REGION Network 2: WatchDog WinCC- PLC
   RUNG wire#powerrail
      Contact( "AlwaysTRUE" )
      Contact( "IEC_Timer_WatchDogWicc-PLC_DB".Q )
      wire#w1
      { S7_Templates := "DestType := Int" } Inc( "Dane_ComunicationControlHMI".tempWatchDog_WinCC )
   END_RUNG
   RUNG wire#powerrail
      Contact( "IEC_Timer_WatchDogWinCC_cd_DB".Q )
   END_RUNG wire#w1
   RUNG wire#powerrail
      { S7_Templates := "SrcType := Int" } GE_Contact(in1 := "Dane_ComunicationControlHMI".tempWatchDog_WinCC, in2 := 70)
      P_Trig( "memRis_Foult_WiCC_PLC" )
      S_Coil( "dbmanagement".sterowanie_1.alarm_comunication_WinCC )
   END_RUNG
   // the same network as SCL:
   IF ("AlwaysTRUE" AND "IEC_Timer_WatchDogWicc-PLC_DB".Q) OR "IEC_Timer_WatchDogWinCC_cd_DB".Q THEN
       "Dane_ComunicationControlHMI".tempWatchDog_WinCC := "Dane_ComunicationControlHMI".tempWatchDog_WinCC + 1;
   END_IF;
   #_w1 := "Dane_ComunicationControlHMI".tempWatchDog_WinCC >= 70;
   #_w2 := #_w1 AND NOT "memRis_Foult_WiCC_PLC";   // rising edge
   "memRis_Foult_WiCC_PLC" := #_w1;
   IF #_w2 THEN "dbmanagement".sterowanie_1.alarm_comunication_WinCC := TRUE; END_IF;
END_REGION
END_FUNCTION_BLOCK

FUNCTION "06_M_active pump selection" : Void   // FC17, LAD
TITLE = Compressor selection from hours
{ S7_Optimized_Access := 'TRUE' }
AUTHOR : rtecmer
VERSION : 0.1
// Ustawienie kolejności wyboru kompresorów z wyrównaniem czasu pracy. Podstawa najmniejsza ilość godzin pracy
// stored: AutoNumber true, IsIECCheckEnabled false, SetENOAutomatically false, UDAEnableTagReadback false
   VAR_IN_OUT
      Reset : Bool;   // Reset po błędzie
   END_VAR
   VAR_TEMP
      tmp_Sum_sek_P1 : Int;
      tmp_Sum_sek_P2 : Int;
      tmp_Sum_sek_P3 : Int;
      tmp_Sum_sek_P4 : Int;
   END_VAR
BEGIN

REGION Network 1: Reakcja na równe liczniki
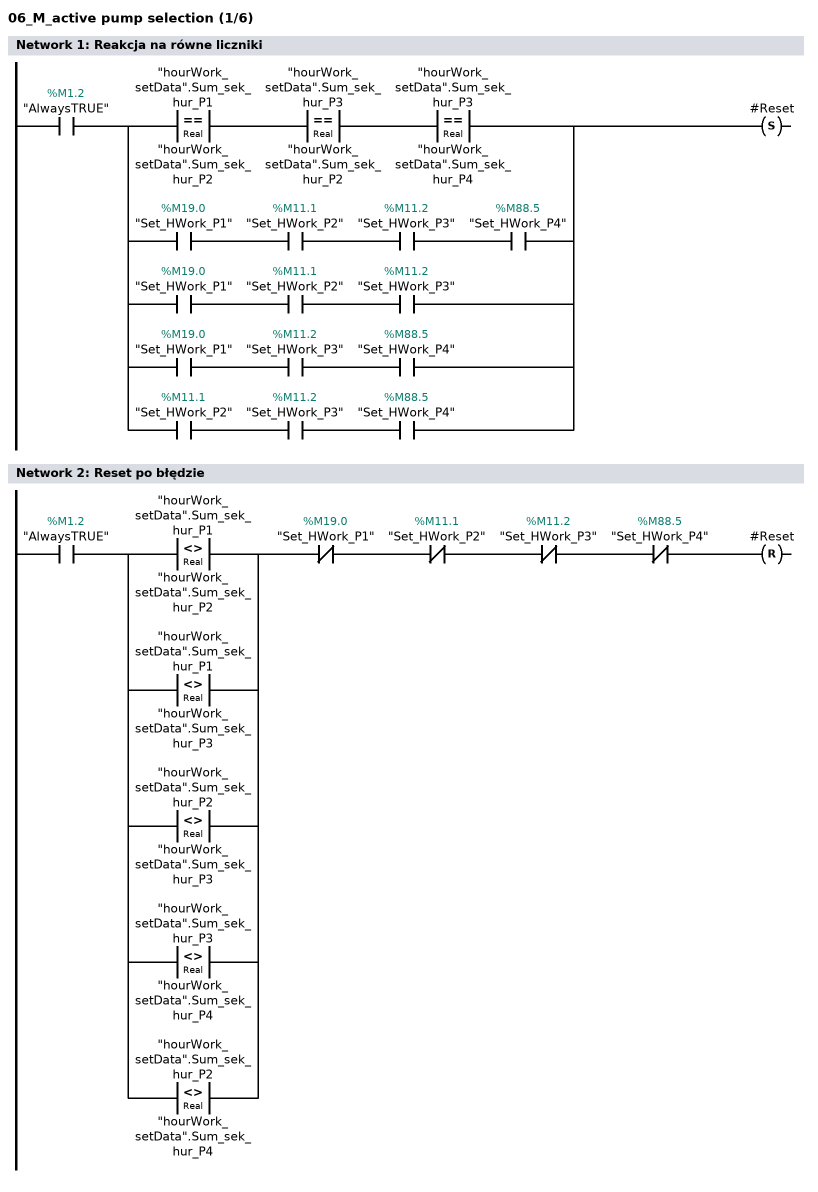
   RUNG wire#powerrail
      Contact( "AlwaysTRUE" )
      wire#w1
      { S7_Templates := "SrcType := Real" } EQ_Contact(in1 := "hourWork_setData".Sum_sek_hur_P1, in2 := "hourWork_setData".Sum_sek_hur_P2)
      { S7_Templates := "SrcType := Real" } EQ_Contact(in1 := "hourWork_setData".Sum_sek_hur_P3, in2 := "hourWork_setData".Sum_sek_hur_P2)
      { S7_Templates := "SrcType := Real" } EQ_Contact(in1 := "hourWork_setData".Sum_sek_hur_P3, in2 := "hourWork_setData".Sum_sek_hur_P4)
      wire#w2
      S_Coil( #Reset )
   END_RUNG
   RUNG wire#w1
      Contact( "Set_HWork_P1" )
      Contact( "Set_HWork_P2" )
      Contact( "Set_HWork_P3" )
      Contact( "Set_HWork_P4" )
   END_RUNG wire#w2
   RUNG wire#w1
      Contact( "Set_HWork_P1" )
      Contact( "Set_HWork_P2" )
      Contact( "Set_HWork_P3" )
   END_RUNG wire#w2
   RUNG wire#w1
      Contact( "Set_HWork_P1" )
      Contact( "Set_HWork_P3" )
      Contact( "Set_HWork_P4" )
   END_RUNG wire#w2
   RUNG wire#w1
      Contact( "Set_HWork_P2" )
      Contact( "Set_HWork_P3" )
      Contact( "Set_HWork_P4" )
   END_RUNG wire#w2
   // the same network as SCL:
   IF "AlwaysTRUE" AND ((("hourWork_setData".Sum_sek_hur_P1 = "hourWork_setData".Sum_sek_hur_P2) AND ("hourWork_setData".Sum_sek_hur_P3 = "hourWork_setData".Sum_sek_hur_P2) AND ("hourWork_setData".Sum_sek_hur_P3 = "hourWork_setData".Sum_sek_hur_P4)) OR ("Set_HWork_P1" AND "Set_HWork_P2" AND "Set_HWork_P3" AND "Set_HWork_P4") OR ("Set_HWork_P1" AND "Set_HWork_P2" AND "Set_HWork_P3") OR ("Set_HWork_P1" AND "Set_HWork_P3" AND "Set_HWork_P4") OR ("Set_HWork_P2" AND "Set_HWork_P3" AND "Set_HWork_P4")) THEN
       #Reset := TRUE;
   END_IF;
END_REGION

REGION Network 2: Reset po błędzie
   RUNG wire#powerrail
      Contact( "AlwaysTRUE" )
      wire#w1
      { S7_Templates := "SrcType := Real" } NE_Contact(in1 := "hourWork_setData".Sum_sek_hur_P1, in2 := "hourWork_setData".Sum_sek_hur_P2)
      wire#w2
      I_Contact( "Set_HWork_P1" )
      I_Contact( "Set_HWork_P2" )
      I_Contact( "Set_HWork_P3" )
      I_Contact( "Set_HWork_P4" )
      R_Coil( #Reset )
   END_RUNG
   RUNG wire#w1
      { S7_Templates := "SrcType := Real" } NE_Contact(in1 := "hourWork_setData".Sum_sek_hur_P1, in2 := "hourWork_setData".Sum_sek_hur_P3)
   END_RUNG wire#w2
   RUNG wire#w1
      { S7_Templates := "SrcType := Real" } NE_Contact(in1 := "hourWork_setData".Sum_sek_hur_P2, in2 := "hourWork_setData".Sum_sek_hur_P3)
   END_RUNG wire#w2
   RUNG wire#w1
      { S7_Templates := "SrcType := Real" } NE_Contact(in1 := "hourWork_setData".Sum_sek_hur_P3, in2 := "hourWork_setData".Sum_sek_hur_P4)
   END_RUNG wire#w2
   RUNG wire#w1
      { S7_Templates := "SrcType := Real" } NE_Contact(in1 := "hourWork_setData".Sum_sek_hur_P2, in2 := "hourWork_setData".Sum_sek_hur_P4)
   END_RUNG wire#w2
   // the same network as SCL:
   IF "AlwaysTRUE" AND (("hourWork_setData".Sum_sek_hur_P1 <> "hourWork_setData".Sum_sek_hur_P2) OR ("hourWork_setData".Sum_sek_hur_P1 <> "hourWork_setData".Sum_sek_hur_P3) OR ("hourWork_setData".Sum_sek_hur_P2 <> "hourWork_setData".Sum_sek_hur_P3) OR ("hourWork_setData".Sum_sek_hur_P3 <> "hourWork_setData".Sum_sek_hur_P4) OR ("hourWork_setData".Sum_sek_hur_P2 <> "hourWork_setData".Sum_sek_hur_P4)) AND NOT "Set_HWork_P1" AND NOT "Set_HWork_P2" AND NOT "Set_HWork_P3" AND NOT "Set_HWork_P4" THEN
       #Reset := FALSE;
   END_IF;
END_REGION

REGION Network 3: Wyłączenie napedów od równych liczników
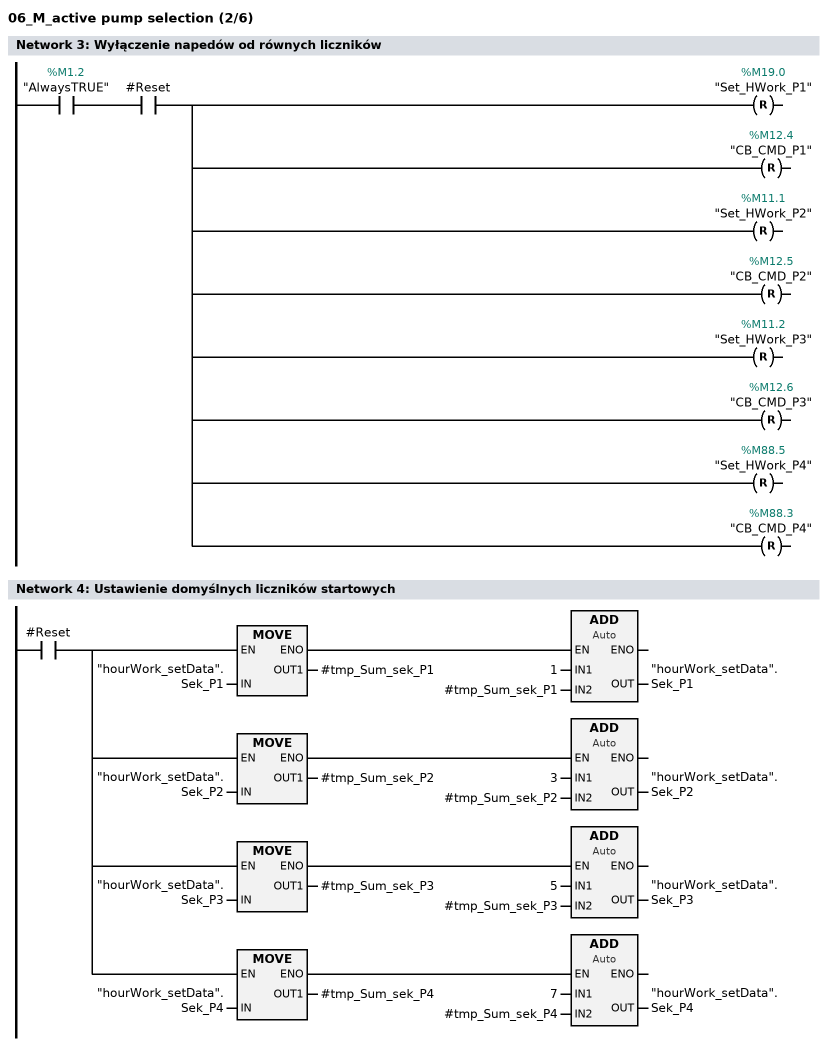
   RUNG wire#powerrail
      Contact( "AlwaysTRUE" )
      Contact( #Reset )
      wire#w1
      R_Coil( "Set_HWork_P1" )
   END_RUNG
   RUNG wire#w1
      R_Coil( "CB_CMD_P1" )
   END_RUNG
   RUNG wire#w1
      R_Coil( "Set_HWork_P2" )
   END_RUNG
   RUNG wire#w1
      R_Coil( "CB_CMD_P2" )
   END_RUNG
   RUNG wire#w1
      R_Coil( "Set_HWork_P3" )
   END_RUNG
   RUNG wire#w1
      R_Coil( "CB_CMD_P3" )
   END_RUNG
   RUNG wire#w1
      R_Coil( "Set_HWork_P4" )
   END_RUNG
   RUNG wire#w1
      R_Coil( "CB_CMD_P4" )
   END_RUNG
   // the same network as SCL:
   IF "AlwaysTRUE" AND #Reset THEN
       "Set_HWork_P1" := FALSE;
       "CB_CMD_P1" := FALSE;
       "Set_HWork_P2" := FALSE;
       "CB_CMD_P2" := FALSE;
       "Set_HWork_P3" := FALSE;
       "CB_CMD_P3" := FALSE;
       "Set_HWork_P4" := FALSE;
       "CB_CMD_P4" := FALSE;
   END_IF;
END_REGION

REGION Network 4: Ustawienie domyślnych liczników startowych
   RUNG wire#powerrail
      Contact( #Reset )
      wire#w1
      Move(in := "hourWork_setData".Sek_P1, out1 => #tmp_Sum_sek_P1)
      Add(in1 := 1, in2 := #tmp_Sum_sek_P1, out => "hourWork_setData".Sek_P1)
   END_RUNG
   RUNG wire#w1
      Move(in := "hourWork_setData".Sek_P2, out1 => #tmp_Sum_sek_P2)
      Add(in1 := 3, in2 := #tmp_Sum_sek_P2, out => "hourWork_setData".Sek_P2)
   END_RUNG
   RUNG wire#w1
      Move(in := "hourWork_setData".Sek_P3, out1 => #tmp_Sum_sek_P3)
      Add(in1 := 5, in2 := #tmp_Sum_sek_P3, out => "hourWork_setData".Sek_P3)
   END_RUNG
   RUNG wire#w1
      Move(in := "hourWork_setData".Sek_P4, out1 => #tmp_Sum_sek_P4)
      Add(in1 := 7, in2 := #tmp_Sum_sek_P4, out => "hourWork_setData".Sek_P4)
   END_RUNG
   // the same network as SCL:
   IF #Reset THEN
       #tmp_Sum_sek_P1 := "hourWork_setData".Sek_P1;
       "hourWork_setData".Sek_P1 := 1 + #tmp_Sum_sek_P1;
       #tmp_Sum_sek_P2 := "hourWork_setData".Sek_P2;
       "hourWork_setData".Sek_P2 := 3 + #tmp_Sum_sek_P2;
       #tmp_Sum_sek_P3 := "hourWork_setData".Sek_P3;
       "hourWork_setData".Sek_P3 := 5 + #tmp_Sum_sek_P3;
       #tmp_Sum_sek_P4 := "hourWork_setData".Sek_P4;
       "hourWork_setData".Sek_P4 := 7 + #tmp_Sum_sek_P4;
   END_IF;
END_REGION

REGION Network 5: Znacznik wyrównywania czasu pracy z falownika dla P1
   // bit tryb automat P1
   // Jesli najmniej godzin pracy to usta znacznik.
   // Ale bierz po uwagę czy kompresor P1 , P4 już nie pracuje lub nie jest w trybie automat.
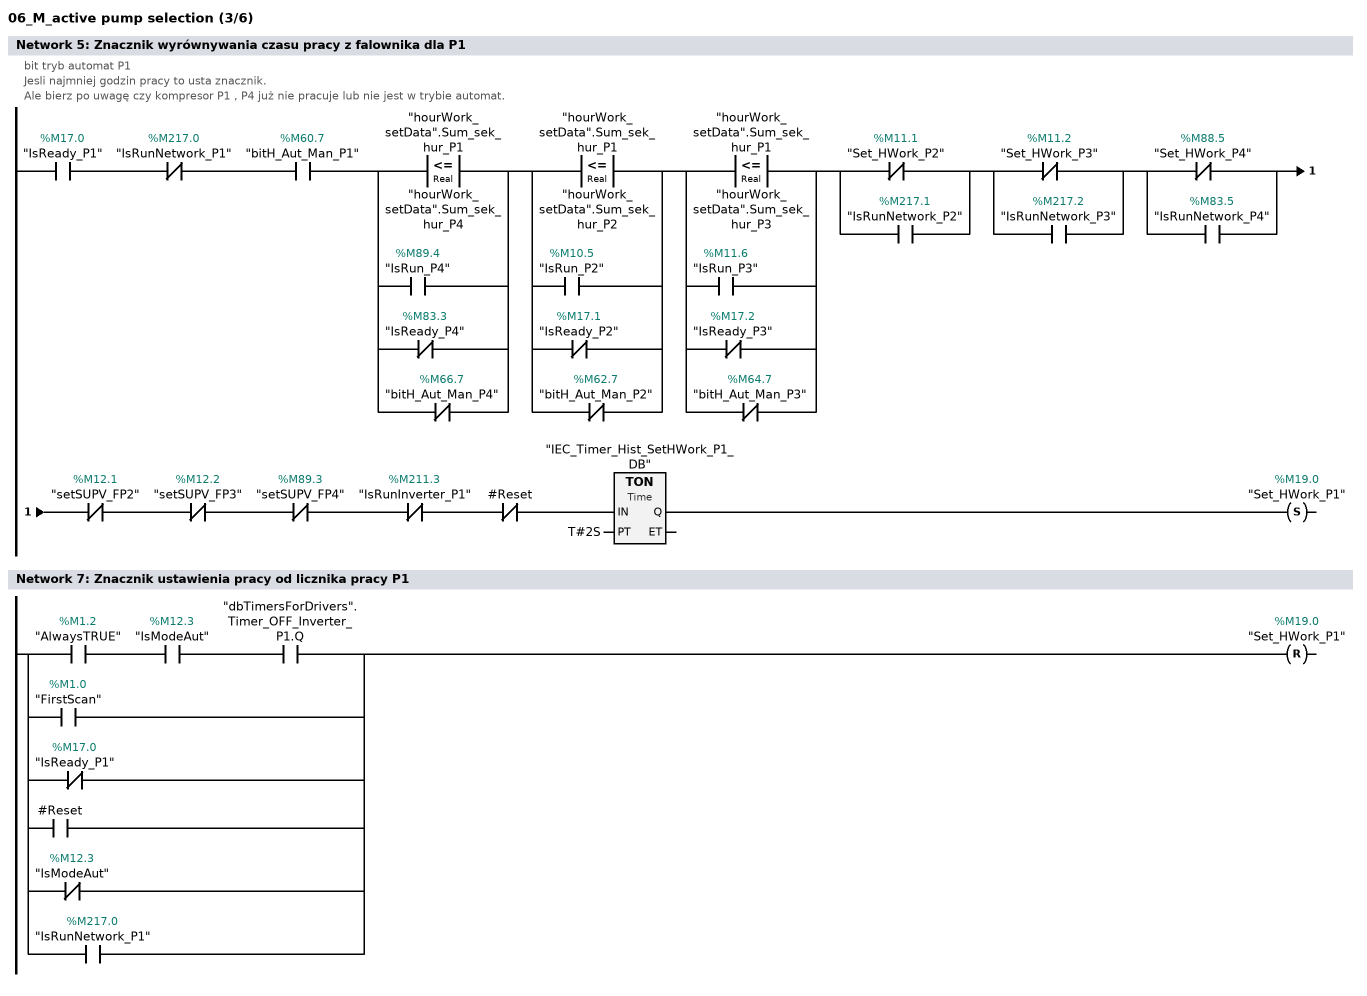
   RUNG wire#powerrail
      Contact( "IsReady_P1" )
      I_Contact( "IsRunNetwork_P1" )
      Contact( "bitH_Aut_Man_P1" )
      wire#w1
      { S7_Templates := "SrcType := Real" } LE_Contact(in1 := "hourWork_setData".Sum_sek_hur_P1, in2 := "hourWork_setData".Sum_sek_hur_P4)
      wire#w2
      { S7_Templates := "SrcType := Real" } LE_Contact(in1 := "hourWork_setData".Sum_sek_hur_P1, in2 := "hourWork_setData".Sum_sek_hur_P2)
      wire#w3
      { S7_Templates := "SrcType := Real" } LE_Contact(in1 := "hourWork_setData".Sum_sek_hur_P1, in2 := "hourWork_setData".Sum_sek_hur_P3)
      wire#w4
      I_Contact( "Set_HWork_P2" )
      wire#w5
      I_Contact( "Set_HWork_P3" )
      wire#w6
      I_Contact( "Set_HWork_P4" )
      wire#w7
      I_Contact( "setSUPV_FP2" )
      I_Contact( "setSUPV_FP3" )
      I_Contact( "setSUPV_FP4" )
      I_Contact( "IsRunInverter_P1" )
      I_Contact( #Reset )
      { S7_Templates := "time_type := Time" } "IEC_Timer_Hist_SetHWork_P1_DB".TON(pt := T#2S, et =>)
      S_Coil( "Set_HWork_P1" )
   END_RUNG
   RUNG wire#w1
      Contact( "IsRun_P4" )
   END_RUNG wire#w2
   RUNG wire#w1
      I_Contact( "IsReady_P4" )
   END_RUNG wire#w2
   RUNG wire#w1
      I_Contact( "bitH_Aut_Man_P4" )
   END_RUNG wire#w2
   RUNG wire#w2
      Contact( "IsRun_P2" )
   END_RUNG wire#w3
   RUNG wire#w2
      I_Contact( "IsReady_P2" )
   END_RUNG wire#w3
   RUNG wire#w2
      I_Contact( "bitH_Aut_Man_P2" )
   END_RUNG wire#w3
   RUNG wire#w3
      Contact( "IsRun_P3" )
   END_RUNG wire#w4
   RUNG wire#w3
      I_Contact( "IsReady_P3" )
   END_RUNG wire#w4
   RUNG wire#w3
      I_Contact( "bitH_Aut_Man_P3" )
   END_RUNG wire#w4
   RUNG wire#w4
      Contact( "IsRunNetwork_P2" )
   END_RUNG wire#w5
   RUNG wire#w5
      Contact( "IsRunNetwork_P3" )
   END_RUNG wire#w6
   RUNG wire#w6
      Contact( "IsRunNetwork_P4" )
   END_RUNG wire#w7
   // the same network as SCL:
   "IEC_Timer_Hist_SetHWork_P1_DB".TON(IN := "IsReady_P1" AND NOT "IsRunNetwork_P1" AND "bitH_Aut_Man_P1" AND (("hourWork_setData".Sum_sek_hur_P1 <= "hourWork_setData".Sum_sek_hur_P4) OR "IsRun_P4" OR NOT "IsReady_P4" OR NOT "bitH_Aut_Man_P4") AND (("hourWork_setData".Sum_sek_hur_P1 <= "hourWork_setData".Sum_sek_hur_P2) OR "IsRun_P2" OR NOT "IsReady_P2" OR NOT "bitH_Aut_Man_P2") AND (("hourWork_setData".Sum_sek_hur_P1 <= "hourWork_setData".Sum_sek_hur_P3) OR "IsRun_P3" OR NOT "IsReady_P3" OR NOT "bitH_Aut_Man_P3") AND (NOT "Set_HWork_P2" OR "IsRunNetwork_P2") AND (NOT "Set_HWork_P3" OR "IsRunNetwork_P3") AND (NOT "Set_HWork_P4" OR "IsRunNetwork_P4") AND NOT "setSUPV_FP2" AND NOT "setSUPV_FP3" AND NOT "setSUPV_FP4" AND NOT "IsRunInverter_P1" AND NOT #Reset,
                           PT := T#2S);
   IF "IEC_Timer_Hist_SetHWork_P1_DB".Q THEN "Set_HWork_P1" := TRUE; END_IF;
END_REGION

REGION Network 6 (SCL): Sprawdzanie czy aktywna w trybie AUT
   IF "Set_HWork_P1" = TRUE AND "bitH_Aut_Man_P1" = FALSE THEN
     // Statement section IF
     "Set_HWork_P1" := FALSE;
     ;
   END_IF;
END_REGION

REGION Network 7: Znacznik ustawienia pracy od licznika pracy P1
   RUNG wire#powerrail
      Contact( "AlwaysTRUE" )
      Contact( "IsModeAut" )
      Contact( "dbTimersForDrivers".Timer_OFF_Inverter_P1.Q )
      wire#w1
      R_Coil( "Set_HWork_P1" )
   END_RUNG
   RUNG wire#powerrail
      Contact( "FirstScan" )
   END_RUNG wire#w1
   RUNG wire#powerrail
      I_Contact( "IsReady_P1" )
   END_RUNG wire#w1
   RUNG wire#powerrail
      Contact( #Reset )
   END_RUNG wire#w1
   RUNG wire#powerrail
      I_Contact( "IsModeAut" )
   END_RUNG wire#w1
   RUNG wire#powerrail
      Contact( "IsRunNetwork_P1" )
   END_RUNG wire#w1
   // the same network as SCL:
   IF ("AlwaysTRUE" AND "IsModeAut" AND "dbTimersForDrivers".Timer_OFF_Inverter_P1.Q) OR "FirstScan" OR NOT "IsReady_P1" OR #Reset OR NOT "IsModeAut" OR "IsRunNetwork_P1" THEN
       "Set_HWork_P1" := FALSE;
   END_IF;
END_REGION

REGION Network 8: Znacznik wyrównywania czasu pracy z falownika dla P2
   // %DB10.DBX9.7 - bit tryb automat P2
   // Jesli najmniej godzin pracy to usta znacznik.
   // Ale bierz po uwagę czy kompresor P1 , P4 już nie pracuje lub nie jest w trybie automat.
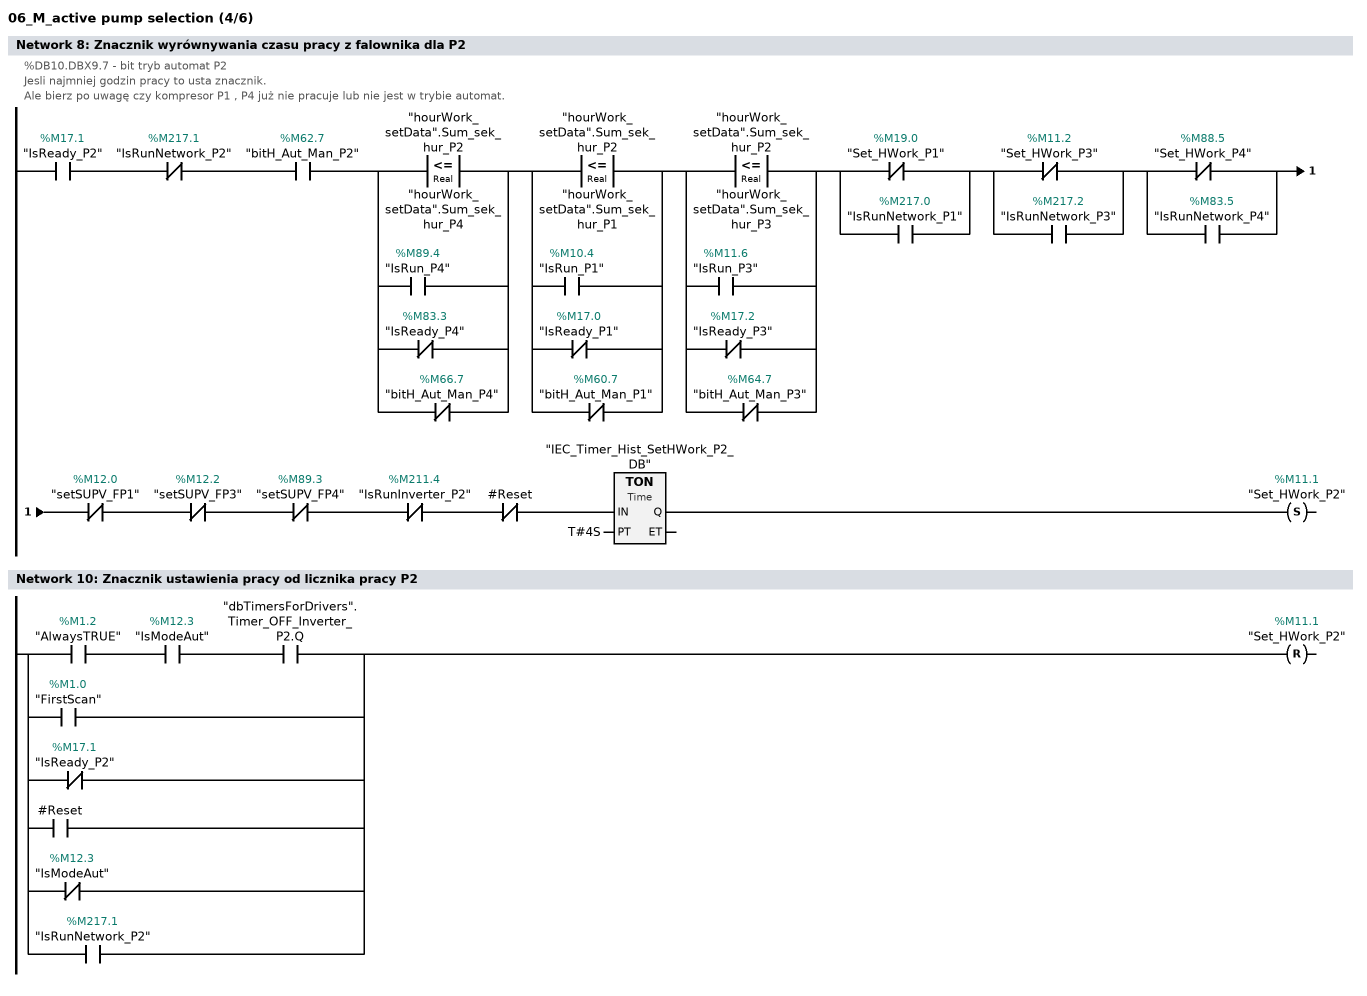
   RUNG wire#powerrail
      Contact( "IsReady_P2" )
      I_Contact( "IsRunNetwork_P2" )
      Contact( "bitH_Aut_Man_P2" )
      wire#w1
      { S7_Templates := "SrcType := Real" } LE_Contact(in1 := "hourWork_setData".Sum_sek_hur_P2, in2 := "hourWork_setData".Sum_sek_hur_P4)
      wire#w2
      { S7_Templates := "SrcType := Real" } LE_Contact(in1 := "hourWork_setData".Sum_sek_hur_P2, in2 := "hourWork_setData".Sum_sek_hur_P1)
      wire#w3
      { S7_Templates := "SrcType := Real" } LE_Contact(in1 := "hourWork_setData".Sum_sek_hur_P2, in2 := "hourWork_setData".Sum_sek_hur_P3)
      wire#w4
      I_Contact( "Set_HWork_P1" )
      wire#w5
      I_Contact( "Set_HWork_P3" )
      wire#w6
      I_Contact( "Set_HWork_P4" )
      wire#w7
      I_Contact( "setSUPV_FP1" )
      I_Contact( "setSUPV_FP3" )
      I_Contact( "setSUPV_FP4" )
      I_Contact( "IsRunInverter_P2" )
      I_Contact( #Reset )
      { S7_Templates := "time_type := Time" } "IEC_Timer_Hist_SetHWork_P2_DB".TON(pt := T#4S, et =>)
      S_Coil( "Set_HWork_P2" )
   END_RUNG
   RUNG wire#w1
      Contact( "IsRun_P4" )
   END_RUNG wire#w2
   RUNG wire#w1
      I_Contact( "IsReady_P4" )
   END_RUNG wire#w2
   RUNG wire#w1
      I_Contact( "bitH_Aut_Man_P4" )
   END_RUNG wire#w2
   RUNG wire#w2
      Contact( "IsRun_P1" )
   END_RUNG wire#w3
   RUNG wire#w2
      I_Contact( "IsReady_P1" )
   END_RUNG wire#w3
   RUNG wire#w2
      I_Contact( "bitH_Aut_Man_P1" )
   END_RUNG wire#w3
   RUNG wire#w3
      Contact( "IsRun_P3" )
   END_RUNG wire#w4
   RUNG wire#w3
      I_Contact( "IsReady_P3" )
   END_RUNG wire#w4
   RUNG wire#w3
      I_Contact( "bitH_Aut_Man_P3" )
   END_RUNG wire#w4
   RUNG wire#w4
      Contact( "IsRunNetwork_P1" )
   END_RUNG wire#w5
   RUNG wire#w5
      Contact( "IsRunNetwork_P3" )
   END_RUNG wire#w6
   RUNG wire#w6
      Contact( "IsRunNetwork_P4" )
   END_RUNG wire#w7
   // the same network as SCL:
   "IEC_Timer_Hist_SetHWork_P2_DB".TON(IN := "IsReady_P2" AND NOT "IsRunNetwork_P2" AND "bitH_Aut_Man_P2" AND (("hourWork_setData".Sum_sek_hur_P2 <= "hourWork_setData".Sum_sek_hur_P4) OR "IsRun_P4" OR NOT "IsReady_P4" OR NOT "bitH_Aut_Man_P4") AND (("hourWork_setData".Sum_sek_hur_P2 <= "hourWork_setData".Sum_sek_hur_P1) OR "IsRun_P1" OR NOT "IsReady_P1" OR NOT "bitH_Aut_Man_P1") AND (("hourWork_setData".Sum_sek_hur_P2 <= "hourWork_setData".Sum_sek_hur_P3) OR "IsRun_P3" OR NOT "IsReady_P3" OR NOT "bitH_Aut_Man_P3") AND (NOT "Set_HWork_P1" OR "IsRunNetwork_P1") AND (NOT "Set_HWork_P3" OR "IsRunNetwork_P3") AND (NOT "Set_HWork_P4" OR "IsRunNetwork_P4") AND NOT "setSUPV_FP1" AND NOT "setSUPV_FP3" AND NOT "setSUPV_FP4" AND NOT "IsRunInverter_P2" AND NOT #Reset,
                           PT := T#4S);
   IF "IEC_Timer_Hist_SetHWork_P2_DB".Q THEN "Set_HWork_P2" := TRUE; END_IF;
END_REGION

REGION Network 9 (SCL): Sprawdzanie czy aktywna w trybie AUT
   IF "Set_HWork_P2" = TRUE AND "bitH_Aut_Man_P2" = FALSE THEN
     // Statement section IF
     "Set_HWork_P2" := FALSE;
     ;
   END_IF;
END_REGION

REGION Network 10: Znacznik ustawienia pracy od licznika pracy P2
   RUNG wire#powerrail
      Contact( "AlwaysTRUE" )
      Contact( "IsModeAut" )
      Contact( "dbTimersForDrivers".Timer_OFF_Inverter_P2.Q )
      wire#w1
      R_Coil( "Set_HWork_P2" )
   END_RUNG
   RUNG wire#powerrail
      Contact( "FirstScan" )
   END_RUNG wire#w1
   RUNG wire#powerrail
      I_Contact( "IsReady_P2" )
   END_RUNG wire#w1
   RUNG wire#powerrail
      Contact( #Reset )
   END_RUNG wire#w1
   RUNG wire#powerrail
      I_Contact( "IsModeAut" )
   END_RUNG wire#w1
   RUNG wire#powerrail
      Contact( "IsRunNetwork_P2" )
   END_RUNG wire#w1
   // the same network as SCL:
   IF ("AlwaysTRUE" AND "IsModeAut" AND "dbTimersForDrivers".Timer_OFF_Inverter_P2.Q) OR "FirstScan" OR NOT "IsReady_P2" OR #Reset OR NOT "IsModeAut" OR "IsRunNetwork_P2" THEN
       "Set_HWork_P2" := FALSE;
   END_IF;
END_REGION

REGION Network 11: Znacznik wyrównywania czasu pracy z falownika P3
   // bit tryb automat P3
   // Jesli najmniej godzin pracy to usta znacznik.
   // Ale bierz po uwagę czy P1, P4 już nie pracuje lub nie jest w trybie automat.
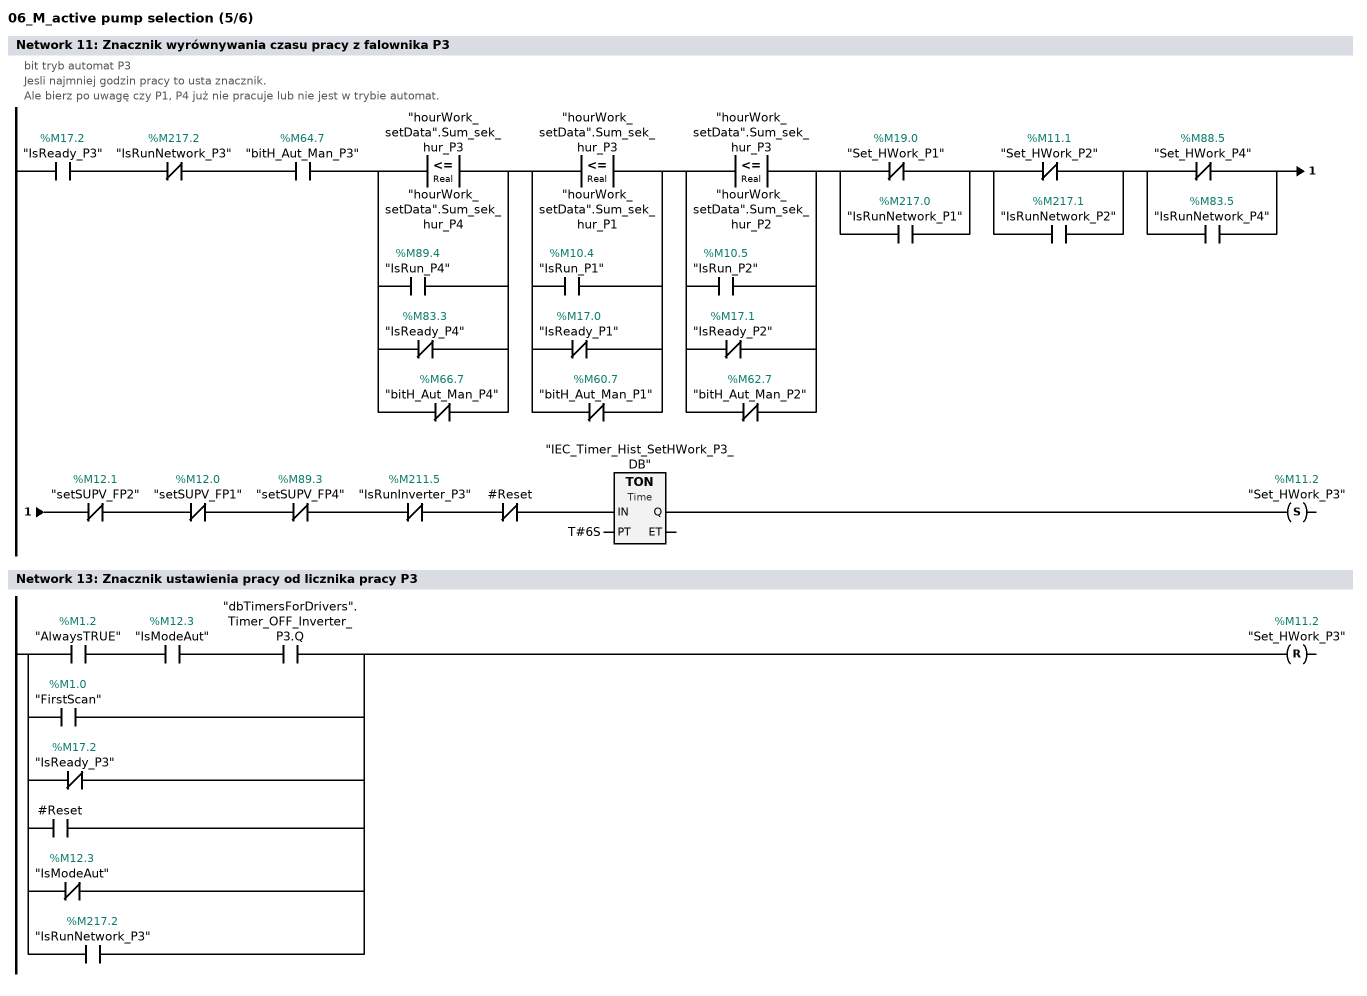
   RUNG wire#powerrail
      Contact( "IsReady_P3" )
      I_Contact( "IsRunNetwork_P3" )
      Contact( "bitH_Aut_Man_P3" )
      wire#w1
      { S7_Templates := "SrcType := Real" } LE_Contact(in1 := "hourWork_setData".Sum_sek_hur_P3, in2 := "hourWork_setData".Sum_sek_hur_P4)
      wire#w2
      { S7_Templates := "SrcType := Real" } LE_Contact(in1 := "hourWork_setData".Sum_sek_hur_P3, in2 := "hourWork_setData".Sum_sek_hur_P1)
      wire#w3
      { S7_Templates := "SrcType := Real" } LE_Contact(in1 := "hourWork_setData".Sum_sek_hur_P3, in2 := "hourWork_setData".Sum_sek_hur_P2)
      wire#w4
      I_Contact( "Set_HWork_P1" )
      wire#w5
      I_Contact( "Set_HWork_P2" )
      wire#w6
      I_Contact( "Set_HWork_P4" )
      wire#w7
      I_Contact( "setSUPV_FP2" )
      I_Contact( "setSUPV_FP1" )
      I_Contact( "setSUPV_FP4" )
      I_Contact( "IsRunInverter_P3" )
      I_Contact( #Reset )
      { S7_Templates := "time_type := Time" } "IEC_Timer_Hist_SetHWork_P3_DB".TON(pt := T#6S, et =>)
      S_Coil( "Set_HWork_P3" )
   END_RUNG
   RUNG wire#w1
      Contact( "IsRun_P4" )
   END_RUNG wire#w2
   RUNG wire#w1
      I_Contact( "IsReady_P4" )
   END_RUNG wire#w2
   RUNG wire#w1
      I_Contact( "bitH_Aut_Man_P4" )
   END_RUNG wire#w2
   RUNG wire#w2
      Contact( "IsRun_P1" )
   END_RUNG wire#w3
   RUNG wire#w2
      I_Contact( "IsReady_P1" )
   END_RUNG wire#w3
   RUNG wire#w2
      I_Contact( "bitH_Aut_Man_P1" )
   END_RUNG wire#w3
   RUNG wire#w3
      Contact( "IsRun_P2" )
   END_RUNG wire#w4
   RUNG wire#w3
      I_Contact( "IsReady_P2" )
   END_RUNG wire#w4
   RUNG wire#w3
      I_Contact( "bitH_Aut_Man_P2" )
   END_RUNG wire#w4
   RUNG wire#w4
      Contact( "IsRunNetwork_P1" )
   END_RUNG wire#w5
   RUNG wire#w5
      Contact( "IsRunNetwork_P2" )
   END_RUNG wire#w6
   RUNG wire#w6
      Contact( "IsRunNetwork_P4" )
   END_RUNG wire#w7
   // the same network as SCL:
   "IEC_Timer_Hist_SetHWork_P3_DB".TON(IN := "IsReady_P3" AND NOT "IsRunNetwork_P3" AND "bitH_Aut_Man_P3" AND (("hourWork_setData".Sum_sek_hur_P3 <= "hourWork_setData".Sum_sek_hur_P4) OR "IsRun_P4" OR NOT "IsReady_P4" OR NOT "bitH_Aut_Man_P4") AND (("hourWork_setData".Sum_sek_hur_P3 <= "hourWork_setData".Sum_sek_hur_P1) OR "IsRun_P1" OR NOT "IsReady_P1" OR NOT "bitH_Aut_Man_P1") AND (("hourWork_setData".Sum_sek_hur_P3 <= "hourWork_setData".Sum_sek_hur_P2) OR "IsRun_P2" OR NOT "IsReady_P2" OR NOT "bitH_Aut_Man_P2") AND (NOT "Set_HWork_P1" OR "IsRunNetwork_P1") AND (NOT "Set_HWork_P2" OR "IsRunNetwork_P2") AND (NOT "Set_HWork_P4" OR "IsRunNetwork_P4") AND NOT "setSUPV_FP2" AND NOT "setSUPV_FP1" AND NOT "setSUPV_FP4" AND NOT "IsRunInverter_P3" AND NOT #Reset,
                           PT := T#6S);
   IF "IEC_Timer_Hist_SetHWork_P3_DB".Q THEN "Set_HWork_P3" := TRUE; END_IF;
END_REGION

REGION Network 12 (SCL): Sprawdzanie czy aktywna w trybie AUT
   IF "Set_HWork_P3" = TRUE AND "bitH_Aut_Man_P3" = FALSE THEN
     // Statement section IF
     "Set_HWork_P3" := FALSE;
     ;
   END_IF;
END_REGION

REGION Network 13: Znacznik ustawienia pracy od licznika pracy P3
   RUNG wire#powerrail
      Contact( "AlwaysTRUE" )
      Contact( "IsModeAut" )
      Contact( "dbTimersForDrivers".Timer_OFF_Inverter_P3.Q )
      wire#w1
      R_Coil( "Set_HWork_P3" )
   END_RUNG
   RUNG wire#powerrail
      Contact( "FirstScan" )
   END_RUNG wire#w1
   RUNG wire#powerrail
      I_Contact( "IsReady_P3" )
   END_RUNG wire#w1
   RUNG wire#powerrail
      Contact( #Reset )
   END_RUNG wire#w1
   RUNG wire#powerrail
      I_Contact( "IsModeAut" )
   END_RUNG wire#w1
   RUNG wire#powerrail
      Contact( "IsRunNetwork_P3" )
   END_RUNG wire#w1
   // the same network as SCL:
   IF ("AlwaysTRUE" AND "IsModeAut" AND "dbTimersForDrivers".Timer_OFF_Inverter_P3.Q) OR "FirstScan" OR NOT "IsReady_P3" OR #Reset OR NOT "IsModeAut" OR "IsRunNetwork_P3" THEN
       "Set_HWork_P3" := FALSE;
   END_IF;
END_REGION

REGION Network 14: Znacznik wyrównywania czasu pracy z falownika P4
   // bit tryb automat P4
   // Jesli najmniej godzin pracy to usta znacznik.
   // Ale bierz po uwagę czy P1, P4 już nie pracuje lub nie jest w trybie automat.
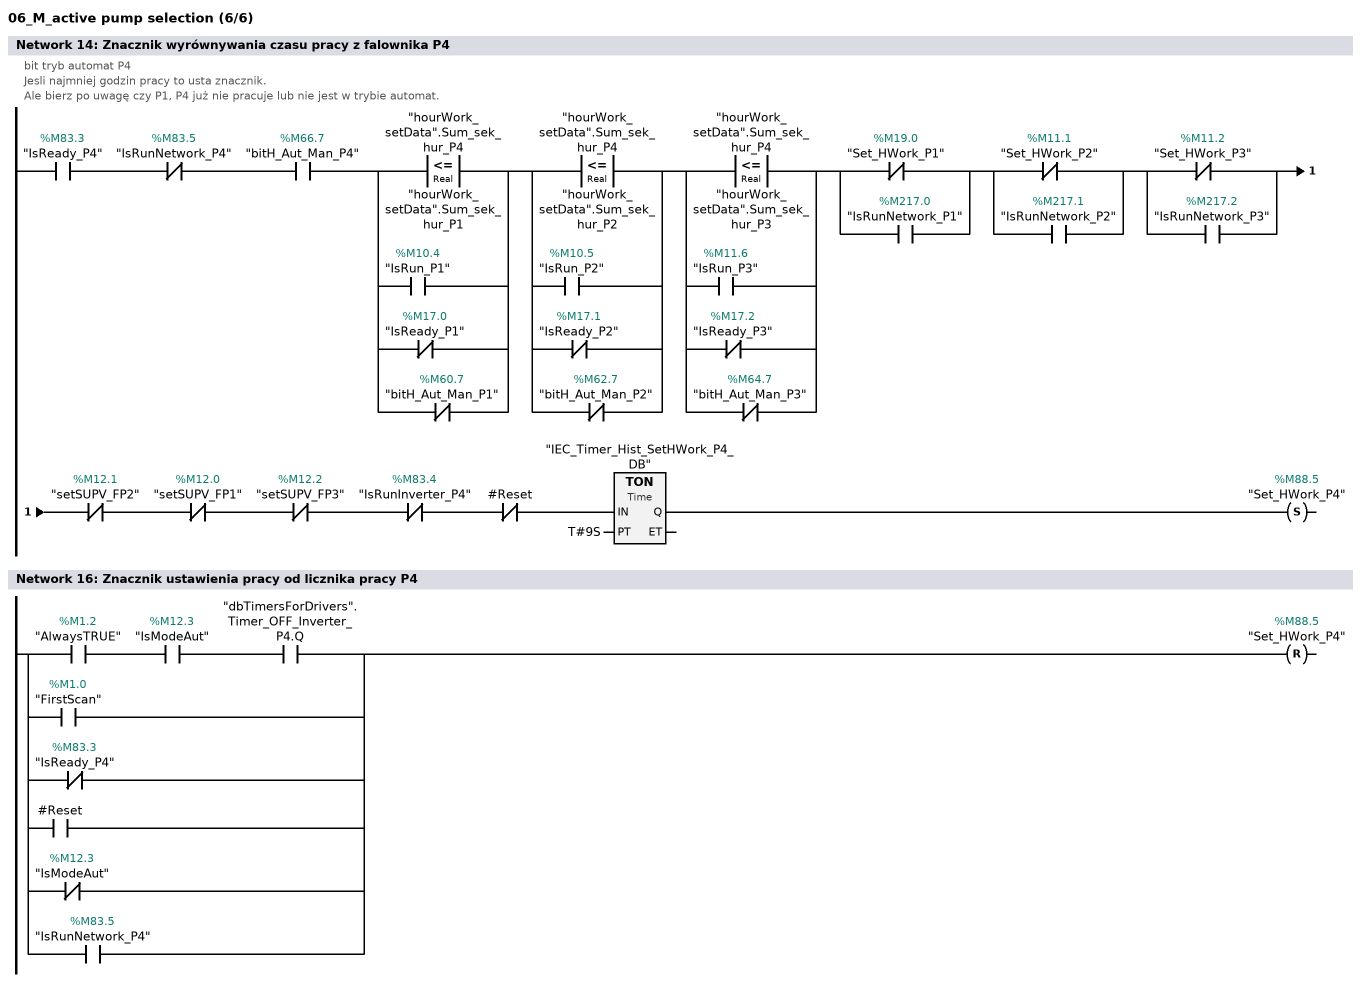
   RUNG wire#powerrail
      Contact( "IsReady_P4" )
      I_Contact( "IsRunNetwork_P4" )
      Contact( "bitH_Aut_Man_P4" )
      wire#w1
      { S7_Templates := "SrcType := Real" } LE_Contact(in1 := "hourWork_setData".Sum_sek_hur_P4, in2 := "hourWork_setData".Sum_sek_hur_P1)
      wire#w2
      { S7_Templates := "SrcType := Real" } LE_Contact(in1 := "hourWork_setData".Sum_sek_hur_P4, in2 := "hourWork_setData".Sum_sek_hur_P2)
      wire#w3
      { S7_Templates := "SrcType := Real" } LE_Contact(in1 := "hourWork_setData".Sum_sek_hur_P4, in2 := "hourWork_setData".Sum_sek_hur_P3)
      wire#w4
      I_Contact( "Set_HWork_P1" )
      wire#w5
      I_Contact( "Set_HWork_P2" )
      wire#w6
      I_Contact( "Set_HWork_P3" )
      wire#w7
      I_Contact( "setSUPV_FP2" )
      I_Contact( "setSUPV_FP1" )
      I_Contact( "setSUPV_FP3" )
      I_Contact( "IsRunInverter_P4" )
      I_Contact( #Reset )
      { S7_Templates := "time_type := Time" } "IEC_Timer_Hist_SetHWork_P4_DB".TON(pt := T#9S, et =>)
      S_Coil( "Set_HWork_P4" )
   END_RUNG
   RUNG wire#w1
      Contact( "IsRun_P1" )
   END_RUNG wire#w2
   RUNG wire#w1
      I_Contact( "IsReady_P1" )
   END_RUNG wire#w2
   RUNG wire#w1
      I_Contact( "bitH_Aut_Man_P1" )
   END_RUNG wire#w2
   RUNG wire#w2
      Contact( "IsRun_P2" )
   END_RUNG wire#w3
   RUNG wire#w2
      I_Contact( "IsReady_P2" )
   END_RUNG wire#w3
   RUNG wire#w2
      I_Contact( "bitH_Aut_Man_P2" )
   END_RUNG wire#w3
   RUNG wire#w3
      Contact( "IsRun_P3" )
   END_RUNG wire#w4
   RUNG wire#w3
      I_Contact( "IsReady_P3" )
   END_RUNG wire#w4
   RUNG wire#w3
      I_Contact( "bitH_Aut_Man_P3" )
   END_RUNG wire#w4
   RUNG wire#w4
      Contact( "IsRunNetwork_P1" )
   END_RUNG wire#w5
   RUNG wire#w5
      Contact( "IsRunNetwork_P2" )
   END_RUNG wire#w6
   RUNG wire#w6
      Contact( "IsRunNetwork_P3" )
   END_RUNG wire#w7
   // the same network as SCL:
   "IEC_Timer_Hist_SetHWork_P4_DB".TON(IN := "IsReady_P4" AND NOT "IsRunNetwork_P4" AND "bitH_Aut_Man_P4" AND (("hourWork_setData".Sum_sek_hur_P4 <= "hourWork_setData".Sum_sek_hur_P1) OR "IsRun_P1" OR NOT "IsReady_P1" OR NOT "bitH_Aut_Man_P1") AND (("hourWork_setData".Sum_sek_hur_P4 <= "hourWork_setData".Sum_sek_hur_P2) OR "IsRun_P2" OR NOT "IsReady_P2" OR NOT "bitH_Aut_Man_P2") AND (("hourWork_setData".Sum_sek_hur_P4 <= "hourWork_setData".Sum_sek_hur_P3) OR "IsRun_P3" OR NOT "IsReady_P3" OR NOT "bitH_Aut_Man_P3") AND (NOT "Set_HWork_P1" OR "IsRunNetwork_P1") AND (NOT "Set_HWork_P2" OR "IsRunNetwork_P2") AND (NOT "Set_HWork_P3" OR "IsRunNetwork_P3") AND NOT "setSUPV_FP2" AND NOT "setSUPV_FP1" AND NOT "setSUPV_FP3" AND NOT "IsRunInverter_P4" AND NOT #Reset,
                           PT := T#9S);
   IF "IEC_Timer_Hist_SetHWork_P4_DB".Q THEN "Set_HWork_P4" := TRUE; END_IF;
END_REGION

REGION Network 15 (SCL): Sprawdzanie czy aktywna w trybie AUT
   IF "Set_HWork_P4" = TRUE AND "bitH_Aut_Man_P4" = FALSE THEN
     // Statement section IF
     "Set_HWork_P4" := FALSE;
     ;
   END_IF;
END_REGION

REGION Network 16: Znacznik ustawienia pracy od licznika pracy P4
   RUNG wire#powerrail
      Contact( "AlwaysTRUE" )
      Contact( "IsModeAut" )
      Contact( "dbTimersForDrivers".Timer_OFF_Inverter_P4.Q )
      wire#w1
      R_Coil( "Set_HWork_P4" )
   END_RUNG
   RUNG wire#powerrail
      Contact( "FirstScan" )
   END_RUNG wire#w1
   RUNG wire#powerrail
      I_Contact( "IsReady_P4" )
   END_RUNG wire#w1
   RUNG wire#powerrail
      Contact( #Reset )
   END_RUNG wire#w1
   RUNG wire#powerrail
      I_Contact( "IsModeAut" )
   END_RUNG wire#w1
   RUNG wire#powerrail
      Contact( "IsRunNetwork_P4" )
   END_RUNG wire#w1
   // the same network as SCL:
   IF ("AlwaysTRUE" AND "IsModeAut" AND "dbTimersForDrivers".Timer_OFF_Inverter_P4.Q) OR "FirstScan" OR NOT "IsReady_P4" OR #Reset OR NOT "IsModeAut" OR "IsRunNetwork_P4" THEN
       "Set_HWork_P4" := FALSE;
   END_IF;
END_REGION
END_FUNCTION

FUNCTION "07_E_drivers Z11 Z12" : Void   // FC30, LAD
TITLE = Driver napedów zasuw Z11, Z12
{ S7_Optimized_Access := 'TRUE' }
AUTHOR : rtecmer
VERSION : 0.1
// Funkcje sterujące napędami w trybie zdalnym, lokalnym
// stored: AutoNumber true, IsIECCheckEnabled false, SetENOAutomatically false, UDAEnableTagReadback false
BEGIN

REGION Network 1: Zasuwa Z11
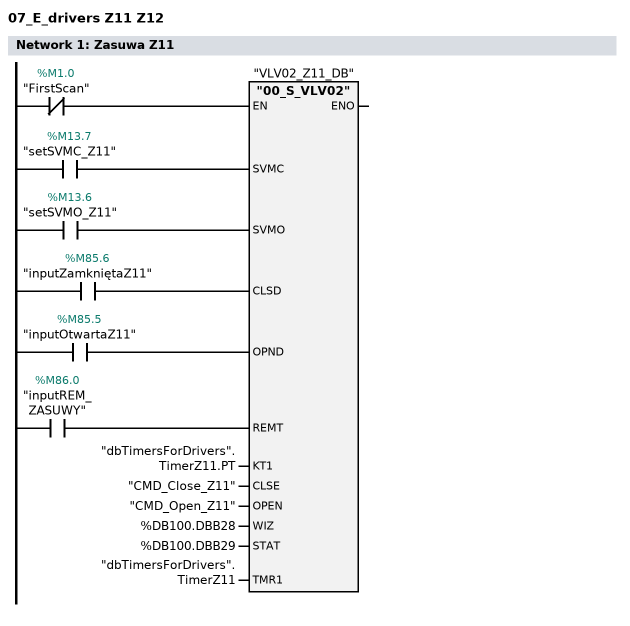
   RUNG wire#powerrail
      I_Contact( "FirstScan" )
      "VLV02_Z11_DB"(SVMC := wire#w1, SVMO := wire#w2, CLSD := wire#w3, OPND := wire#w4, REMT := wire#w5, KT1 := "dbTimersForDrivers".TimerZ11.PT, CLSE := "CMD_Close_Z11", OPEN := "CMD_Open_Z11", WIZ := %DB100.DBB28, STAT := %DB100.DBB29, TMR1 := "dbTimersForDrivers".TimerZ11)
   END_RUNG
   RUNG wire#powerrail
      Contact( "setSVMC_Z11" )
   END_RUNG wire#w1
   RUNG wire#powerrail
      Contact( "setSVMO_Z11" )
   END_RUNG wire#w2
   RUNG wire#powerrail
      Contact( "inputZamkniętaZ11" )
   END_RUNG wire#w3
   RUNG wire#powerrail
      Contact( "inputOtwartaZ11" )
   END_RUNG wire#w4
   RUNG wire#powerrail
      Contact( "inputREM_ZASUWY" )
   END_RUNG wire#w5
   // the same network as SCL:
   IF NOT "FirstScan" THEN
       "VLV02_Z11_DB"(SVMC := "setSVMC_Z11",   // "00_S_VLV02"
                      SVMO := "setSVMO_Z11",
                      CLSD := "inputZamkniętaZ11",
                      OPND := "inputOtwartaZ11",
                      REMT := "inputREM_ZASUWY",
                      KT1 := "dbTimersForDrivers".TimerZ11.PT,
                      CLSE := "CMD_Close_Z11",
                      OPEN := "CMD_Open_Z11",
                      WIZ := %DB100.DBB28,
                      STAT := %DB100.DBB29,
                      TMR1 := "dbTimersForDrivers".TimerZ11);
   END_IF;
END_REGION
END_FUNCTION

ORGANIZATION_BLOCK "Cyclic interrupt_1"
{ S7_Optimized_Access := 'TRUE' }
VERSION : 0.1

BEGIN
	(*
	//=============================================================================
	//(JZWiK S.A Radosław Tecmer)
	//(c)Copyright (2021) All Rights Reserved
	//-----------------------------------------------------------------------------
	//Testowane z:   (system docelowy z  FW 4.4)
	//Pakiet inżynierski:   TIA Portal (V14 Sp1 Update 9)
	//Ograniczenia:  ( - )
	//Wymagania:  (minimalne S7-1200 CPU 1215C FW 4.2 .)
	//Funkcjonalnośc: (Pobranie wartości z wejść analogowych )
	//-----------------------------------------------------------------------------
	//Zmainy wprowadzone:
	//Wersja  Data       Osoba wprowadzająca zmiany - ekspert
	//01.00.00 11.01.2022 (Tecmer Radosław - twórca) Pieresza wersja 01.00.00
	//=============================================================================
	*)
	// Analogi 
	// ciśnienie przetłaczania miasto 
	"dbdane".PV_analaog_B6 := "IW64":P;
	// ciśnienie magistrala
	"dbdane".PV_analaog_B7 := "IW66":P;
	
	//zbiornik nr 3
	"dbdane".actSignalTank3 := "IW164":P;
	
	// poziom w zbiorniku 1
	"dbdane".actSignalTank1:= "IW68":P;
	
	//poziom w zbiorniku 2
	"dbdane".actSignalTank2:= "IW70":P;
END_ORGANIZATION_BLOCK

FUNCTION "00_S_SclScaleLinearRealToInt" : Int
{ S7_Optimized_Access := 'TRUE' }
VERSION : 0.1
   VAR_INPUT 
      x : Real;
      yMin : Int;
      yMax : Int;
      x0 : Real;
      y0 : Int;
      x1 : Real;
      y1 : Int;
   END_VAR

   VAR_TEMP 
      tempY0real : Real;
      tempY1real : Real;
      tempYreal : Real;
      tempYminReal : Real;
      tempYmaxReal : Real;
   END_VAR


BEGIN
	#tempY0real := INT_TO_REAL(#y0);
	#tempY1real := INT_TO_REAL(#y1);
	#tempYminReal := INT_TO_REAL(#yMin);
	#tempYmaxReal := INT_TO_REAL(#yMax);
	
	IF (#y1 - #y0) = 0 OR (#x1 - #x0) = 0 OR (#x - #x0) = 0 OR #yMin > #yMax
	THEN
	    #"00_S_SclScaleLinearRealToInt" := 0;
	ELSE
	    #tempYreal := (#tempY1real - #tempY0real) / (#x1 - #x0) * (#x - #x0) + #tempY0real;
	END_IF;
	
	IF #tempYreal < #tempYminReal THEN
	    #"00_S_SclScaleLinearRealToInt" := 0;
	ELSIF #tempYreal > #tempYmaxReal THEN
	    #"00_S_SclScaleLinearRealToInt" := #yMax;
	ELSE
	    #"00_S_SclScaleLinearRealToInt" := REAL_TO_INT(#tempYreal);
	END_IF;
END_FUNCTION

FUNCTION "05_S_variables_dbModbusMaster_1" : Void
{ S7_Optimized_Access := 'TRUE' }
AUTHOR : RTecmer
FAMILY : 'HMI(XM)'
VERSION : 0.1
//Przekazywanie zmiennych między urządzeniami

BEGIN
	(*
	//=============================================================================
	//(JZWiK S.A Radosław Tecmer)
	//(c)Copyright (2021) All Rights Reserved
	//-----------------------------------------------------------------------------
	//Testowane z:   (system docelowy z  FW 4.2)
	//Pakiet inżynierski:   TIA Portal (V14 Sp1 Update 9)
	//Ograniczenia:  ( - )
	//Wymagania:  (minimalne S7-1200 CPU 1214 FW 3.2 .)
	//Funkcjonalnośc: (Kopiowanie bloków danych między blokiem danych Modbus -SCADA  )
	//-----------------------------------------------------------------------------
	//Zmainy wprowadzone:
	//Wersja  Data       Osoba wprowadzająca zmiany - ekspert
	//01.00.00 17.11.2021 (Tecmer Radosław - twórca) Pieresza wersja 01.00.00
	//=============================================================================
	*)
	
	REGION Analogi
	  // 
	
	  
	  
	END_REGION
	
	
	
	
	
	 
	
	
	
	
	
	
	
	
	
	
	
	
	
	
	
	
	
	
	
	
	
	
END_FUNCTION

FUNCTION "06_M_Write_to DB_HoldReg_MT101" : Void
{ S7_Optimized_Access := 'TRUE' }
AUTHOR : rtecmer
VERSION : 0.1

BEGIN
	(*
	//=============================================================================
	//(JZWiK S.A Radosław Tecmer)
	//(c)Copyright (2021) All Rights Reserved
	//-----------------------------------------------------------------------------
	//Testowane z:   (system docelowy z  FW 4.2)
	//Pakiet inżynierski:   TIA Portal (V14 Sp1 Update 9)
	//Ograniczenia:  ( - )
	//Wymagania:  (minimalne S7-1200 CPU 1214 FW 3.2 .)
	//Funkcjonalnośc: (Kopiowanie bloków danych )
	//-----------------------------------------------------------------------------
	//Zmainy wprowadzone:
	//Wersja  Data       Osoba wprowadzająca zmiany - ekspert
	//01.00.00 17.11.2021 (Tecmer Radosław - twórca) Pieresza wersja 01.00.00
	//=============================================================================
	*)
	
	
	
	REGION  Stacja Zasów Status Napędów
	  // PLC Zasówy z modbus TCP
	  "db10datablock".instvValveZ1 := "db10datablock".instvValveZ1;
	
	  
	  // Do instancji SCADA na MT101
	  "dbHoldRegSlave_to_MT101".instvValveZ1 := "db10datablock".instvValveZ1;
	
	  
	END_REGION
	
	
	
	REGION Analogi
	  // Przekazanie
	  "dbHoldRegSlave_to_MT101".instB5bar_act := "db10datablock".instB5_bar_act_magistrala;
	  "dbHoldRegSlave_to_MT101".instB6bar_act := "db10datablock".instB6_bar_act_miasto;
	  "dbHoldRegSlave_to_MT101".instB7bar_act := "db10datablock".instB7_bar_act_pompownia;
	  "dbHoldRegSlave_to_MT101".instB8bar_act := "dbdane".act_Value_B8;
	  "dbHoldRegSlave_to_MT101".instFlowDN225_act := "db10datablock".instFlowDN225_act_Q1;
	  "dbHoldRegSlave_to_MT101".instFlowDN225_sum := "db10datablock".instSumFlowDN225_Q1;
	  "dbHoldRegSlave_to_MT101".instFlowDN500_act := "db10datablock".instFlowDN500_act_Q2;
	  "dbHoldRegSlave_to_MT101".instFlowDN500_sum := "db10datablock".instSumFlowDN500_Q2;
	  "dbHoldRegSlave_to_MT101".instCurrent_Inverter := REAL_TO_INT("db10datablock".inst_act_Current_Inverters);
	  "dbHoldRegSlave_to_MT101".instHz_Inverter := REAL_TO_INT("db10datablock".act_Hz_Inverter_1);
	  
	
	  // Miasto DN225
	  // aktualny
	  
	  "dbHoldRegSlave_to_MT101".instFlowDN225_act := "dbModbusRTU_Reg"."Przepływomierz nr1 pompownia".ID6_przeływu_VF_Adres_0;
	  //Suma
	  "dbHoldRegSlave_to_MT101".instFlowDN225_sum := "dbModbusRTU_Reg"."Przepływomierz nr1 pompownia".ID6_objętość_VF_Adres_2;
	END_REGION
	
	
	
	
	
	
	
	
	
END_FUNCTION

FUNCTION_BLOCK "06_S_FindPumpWithMinWorkTime"
TITLE = FindPumpWithMinWorkTime
{ S7_Optimized_Access := 'TRUE' }
AUTHOR : rtecmer
VERSION : 0.1
//Funkcja poszukuje pompy z najniższym licznikiem
   VAR_IN_OUT 
      chosenPump : Int;   // wybrana pompa numer
   END_VAR

   VAR 
      minTime : Real;   // mniejszy licznik
   END_VAR


BEGIN
	(*
	//=============================================================================
	//(JZWiK S.A Radosław Tecmer)
	//(c)Copyright (2021) All Rights Reserved
	//-----------------------------------------------------------------------------
	//Testowane z:   (system docelowy z  FW 4.4)
	//Pakiet inżynierski:   TIA Portal (V14 Sp1 Update 9)
	//Ograniczenia:  ( - )
	//Wymagania:  (minimalne S7-1200 CPU 1215C FW 4.2 .)
	//Funkcjonalnośc: (Funkcja poszukuje pompy z najniższym stanem licznika pracy 
	//                  wcelu sterowania wyrównywaniem czasu pracy napedów. 
	//                  Przekazuje do bloku danych wcelu udostępnienia funkcji
	//                  SetActivePump.)
	//-----------------------------------------------------------------------------
	//Zmainy wprowadzone:
	//Wersja  Data       Osoba wprowadzająca zmiany - ekspert
	//01.00.00 23.08.2023 (Tecmer Radosław - twórca) Pieresza wersja 01.00.00
	//=============================================================================
	*)
	
	// inicjacja wartości począdkowej maksymalnej
	#minTime := 2147483647;
	// zerowanie zmiennej
	#chosenPump := 0;
	
	IF "IsReady_P1" AND "bitH_Aut_Man_P1"AND ("IsRunNetwork_P1" = FALSE) AND "TurnOffPump"<> 1 THEN
	  IF "hourWork_setData".Sum_sek_hur_P1 < #minTime THEN
	    #minTime := "hourWork_setData".Sum_sek_hur_P1;
	    #chosenPump := 1;
	  END_IF;
	END_IF;
	
	IF "IsReady_P2" AND "bitH_Aut_Man_P2" AND ("IsRunNetwork_P2" = FALSE) AND "TurnOffPump" <> 2 THEN
	  IF "hourWork_setData".Sum_sek_hur_P2 < #minTime THEN
	    #minTime := "hourWork_setData".Sum_sek_hur_P2;
	    #chosenPump := 2;
	  END_IF;
	END_IF;
	
	IF "IsReady_P3" AND "bitH_Aut_Man_P3" AND ("IsRunNetwork_P3" = FALSE) AND "TurnOffPump" <> 3 THEN
	  IF "hourWork_setData".Sum_sek_hur_P3 < #minTime THEN
	    #minTime := "hourWork_setData".Sum_sek_hur_P3;
	    #chosenPump := 3;
	  END_IF;
	END_IF;
	
	IF "IsReady_P4" AND "bitH_Aut_Man_P4" AND ("IsRunNetwork_P4" = FALSE) AND "TurnOffPump" <> 4 THEN
	  IF "hourWork_setData".Sum_sek_hur_P4 < #minTime THEN
	    #minTime := "hourWork_setData".Sum_sek_hur_P4;
	    #chosenPump := 4;
	  END_IF;
	END_IF;
	
	
	// kontrola czy nie ma załączonej pompy z sieci w wypadku braku wskazanej wiodacej
	// jeśli tak to wyłącz
	IF #chosenPump = 0 THEN
	  // Sprawdz czy jakiaś pracuje na sieci
	  IF "IsRunNetwork_P1" = TRUE THEN
	    // Statement section IF
	    "setCMD_SP1" := FALSE;
	    ;
	  END_IF;
	  IF "IsRunNetwork_P2" = TRUE THEN
	    // Statement section IF
	    "setCMD_SP2" := FALSE;
	    ;
	  END_IF;
	  IF "IsRunNetwork_P3" = TRUE THEN
	    // Statement section IF
	    "setCMD_SP3" := FALSE;
	    ;
	  END_IF;
	  
	  ;
	END_IF;
	
	
	
	RETURN;
	
END_FUNCTION_BLOCK

FUNCTION_BLOCK "06_S_SetActivePump"
TITLE = SetActivePump 
{ S7_Optimized_Access := 'TRUE' }
AUTHOR : rtecmer
VERSION : 0.1
//Funkacja ustawia aktywną pompę do pracy jak wiodąca na podstawie czasu pracy. Funkcja pozwala na wrównywanie liczników pracy
   VAR_IN_OUT 
      ActivePump : Int;   // numer aktywnej pompy - wiodącej
      pumpNum : Int;
   END_VAR


BEGIN
	(*
	//=============================================================================
	//(JZWiK S.A Radosław Tecmer)
	//(c)Copyright (2021) All Rights Reserved
	//-----------------------------------------------------------------------------
	//Testowane z:   (system docelowy z  FW 4.4)
	//Pakiet inżynierski:   TIA Portal (V14 Sp1 Update 9)
	//Ograniczenia:  ( - )
	//Wymagania:  (minimalne S7-1200 CPU 1215C FW 4.2 .)
	//Funkcjonalnośc: (Funkcja ustawia wskazany znacznik Set_HWork_Px 
	//                 jesli spełnione są warunki aktywując pompę wiodącą)
	//-----------------------------------------------------------------------------
	//Zmainy wprowadzone:
	//Wersja  Data       Osoba wprowadzająca zmiany - ekspert
	//01.00.00 23.09.2023 (Tecmer Radosław - twórca) Pieresza wersja 01.00.00
	//=============================================================================
	*)
	
	
	  "Set_HWork_P1" := FALSE;
	  "Set_HWork_P2" := FALSE;
	  "Set_HWork_P3" := FALSE;
	  "Set_HWork_P4" := FALSE;
	
	//"setSUPV_FP2"
	
	// zmiena "dbdane".chosenPump  przekazana z funkcji "FindPumpWithMinWorkTime" 
	CASE "dbdane".chosenPump OF
	  1:
	    IF "IsReady_P1" AND "bitH_Aut_Man_P1" AND ("IsRunInverter_P1" = FALSE) AND "IsRunInverter_P1" = FALSE THEN
	      "Set_HWork_P1" := TRUE;
	      #ActivePump := 1;
	    END_IF;
	  2:
	    IF "IsReady_P2" AND "bitH_Aut_Man_P2"AND ("IsRunInverter_P2" = FALSE) AND "IsRunInverter_P2" = FALSE THEN
	      "Set_HWork_P2" := TRUE;
	      #ActivePump := 2;
	    END_IF;
	  3:
	    IF "IsReady_P3" AND "bitH_Aut_Man_P3" AND ("IsRunInverter_P3" = FALSE) AND "IsRunInverter_P3" = FALSE THEN
	      "Set_HWork_P3" := TRUE;
	      #ActivePump := 3;
	    END_IF;
	  4:
	    IF "IsReady_P4" AND "bitH_Aut_Man_P4" AND ("IsRunInverter_P4" = FALSE) AND "IsRunInverter_P4" = FALSE THEN
	      "Set_HWork_P4" := TRUE;
	      #ActivePump := 4;
	    END_IF;
	  ELSE
	    // W przypadku niepoprawnej wartości pumpNum, wyłącz wszystkie pompy
	    "Set_HWork_P1" := FALSE;
	    "Set_HWork_P2":= FALSE;
	    "Set_HWork_P3" := FALSE;
	    "Set_HWork_P4" := FALSE;
	END_CASE;
	
	// Aktualizacja zmiennej globalnej
	#pumpNum := "dbdane".chosenPump;
	#ActivePump := #pumpNum;
	
	
END_FUNCTION_BLOCK

DATA_BLOCK "01_E_PID_Reset_DB"   // DB83
AUTHOR : rtecmer
VERSION : 0.1
// stored: AutoNumber true, DBAccessibleFromOPCUA true, InstanceOfName 01_E_PID_Reset, InstanceOfType FB
"01_E_PID_Reset"
BEGIN
END_DATA_BLOCK

DATA_BLOCK "01_E_cleaning_the_alarm_reset_button_DB"   // DB48
AUTHOR : rtecme
VERSION : 0.1
// stored: AutoNumber true, DBAccessibleFromOPCUA true, InstanceOfName 01_E_cleaning_the_alarm_reset_button, InstanceOfType FB
"01_E_cleaning_the_alarm_reset_button"
BEGIN
END_DATA_BLOCK

DATA_BLOCK "04_A_Out_analog_DB"   // DB85
AUTHOR : rtecmer
VERSION : 0.1
// stored: AutoNumber true, DBAccessibleFromOPCUA true, InstanceOfName 04_A_Out_analog, InstanceOfType FB
"04_A_Out_analog"
BEGIN
END_DATA_BLOCK

DATA_BLOCK "06_M_control strategy Z11semi-automatic_DB"   // DB150
AUTHOR : rtecmer
VERSION : 0.1
// stored: AutoNumber true, DBAccessibleFromOPCUA true, InstanceOfName 06_M_control strategy Z11, InstanceOfType FB
"06_M_control strategy Z11"
BEGIN
END_DATA_BLOCK

DATA_BLOCK "MainControlSetPump_DB"   // DB99
AUTHOR : vrtecmer
VERSION : 0.1
// stored: AutoNumber true, DBAccessibleFromOPCUA true, InstanceOfName MainControlSetPump, InstanceOfType FB
"MainControlSetPump"
   // VAR_IN_OUT
   //    chosenPump : Int;
   // END_VAR
BEGIN
END_DATA_BLOCK

DATA_BLOCK "FindPumpWithMinWorkTime_DB_1"   // DB87
AUTHOR : rtecmer
VERSION : 0.1
// stored: AutoNumber true, DBAccessibleFromOPCUA true, InstanceOfName FindPumpWithMinWorkTime, InstanceOfType FB
"FindPumpWithMinWorkTime"
   // VAR_IN_OUT
   //    chosenPump : Int;
   // END_VAR
   // VAR
   //    minTime : Real;
   // END_VAR
BEGIN
END_DATA_BLOCK

DATA_BLOCK "SetActivePump_DB_1"   // DB86
AUTHOR : rtecmer
VERSION : 0.1
// stored: AutoNumber true, DBAccessibleFromOPCUA true, InstanceOfName SetActivePump, InstanceOfType FB
"SetActivePump"
   // VAR_IN_OUT
   //    ActivePump : Int;
   //    pumpNum : Int;
   // END_VAR
BEGIN
END_DATA_BLOCK

DATA_BLOCK "EX012_IDB8_ErrorHandling"   // DB104
VERSION : 0.1
// stored: AutoNumber false, DBAccessibleFromOPCUA true, InstanceOfName EX012_ErrorHandling, InstanceOfType FB
"EX012_ErrorHandling"
   // VAR_INPUT
   //    LED : Int;
   //    CounterError : USInt;
   // END_VAR
   // VAR_OUTPUT
   //    RedLED : Bool;
   // END_VAR
   // VAR
   //    tempCounterDiagStatus : USInt;
   //    tempCounterError : USInt;
   // END_VAR
BEGIN
END_DATA_BLOCK

DATA_BLOCK "alarm_min_DN500_B5_DB"   // DB19
AUTHOR : rt69
VERSION : 0.1
// stored: AutoNumber true, DBAccessibleFromOPCUA true, InstanceOfName 01_E_Alarm_min_bar_empty_tanks, InstanceOfType FB
"01_E_Alarm_min_bar_empty_tanks"
BEGIN
END_DATA_BLOCK

DATA_BLOCK "alarmpump_value_press"   // DB143
AUTHOR : rtecmer
VERSION : 0.1
// stored: AutoNumber true, DBAccessibleFromOPCUA true, InstanceOfName 06_M_Alarm-Pomps_value_press, InstanceOfType FB
"06_M_Alarm-Pomps_value_press"
BEGIN
END_DATA_BLOCK

DATA_BLOCK "AutomaticPIDReset_DB"   // DB21
VERSION : 0.1
// stored: AutoNumber true, DBAccessibleFromOPCUA true, InstanceOfName 00_S_AutomaticPIDReset, InstanceOfType FB
"00_S_AutomaticPIDReset"
BEGIN
END_DATA_BLOCK

DATA_BLOCK "Control Current Overload_DB"   // DB72
AUTHOR : rtecmer
VERSION : 0.1
// stored: AutoNumber true, DBAccessibleFromOPCUA true, InstanceOfName 01_E_Inverter current overload control, InstanceOfType FB
"01_E_Inverter current overload control"
BEGIN
END_DATA_BLOCK

DATA_BLOCK "Strategia sterowaia Z11_DB_1"   // DB146
AUTHOR : rtecmer
VERSION : 0.1
// stored: AutoNumber true, DBAccessibleFromOPCUA true, InstanceOfName 06_M_control strategy Z11, InstanceOfType FB
"06_M_control strategy Z11"
BEGIN
END_DATA_BLOCK

DATA_BLOCK "dbModbus_falownik_konwersja"   // DB7
AUTHOR : rtecmer
VERSION : 0.1
// stored: AutoNumber true, DBAccessibleFromOPCUA true, InstanceOfName 08_M_Converting parameters from the inverter, InstanceOfType FB
"08_M_Converting parameters from the inverter"
BEGIN
END_DATA_BLOCK

DATA_BLOCK "FB220_TimeSyn_PLC_To_HMI_DB_1"   // DB78
VERSION : 0.1
// stored: AutoNumber true, DBAccessibleFromOPCUA true, InstanceOfName 02_R_TimeSyn_PLC_To_HMI, InstanceOfType FB
"02_R_TimeSyn_PLC_To_HMI"
BEGIN
END_DATA_BLOCK

DATA_BLOCK "VLV02_Z11_DB"   // DB24
AUTHOR : RTecmer
VERSION : 0.2
// stored: AutoNumber true, DBAccessibleFromOPCUA true, InstanceOfName 00_S_VLV02, InstanceOfType FB
"00_S_VLV02"
BEGIN
END_DATA_BLOCK

DATA_BLOCK "VLV02_Z12_DB"   // DB80
AUTHOR : RTecmer
VERSION : 0.2
// stored: AutoNumber true, DBAccessibleFromOPCUA true, InstanceOfName 00_S_VLV02, InstanceOfType FB
"00_S_VLV02"
BEGIN
END_DATA_BLOCK

DATA_BLOCK "Byte Status Z11 Z12_DB"   // DB82
AUTHOR : rtecmer
VERSION : 0.1
// stored: AutoNumber true, DBAccessibleFromOPCUA true, InstanceOfName 06_M_Byte status Z11 Z12, InstanceOfType FB
"06_M_Byte status Z11 Z12"
BEGIN
END_DATA_BLOCK

DATA_BLOCK "F_TRIG_DB_przechwycenie_powrotu_bar_valueTanks"   // DB112
// stored: AutoNumber true, DBAccessibleFromOPCUA true, InstanceOfName F_TRIG, OfSystemLibElement F_TRIG, OfSystemLibVersion 1.0
"F_TRIG"
   // VAR_INPUT
   //    CLK : Bool;
   // END_VAR
   // VAR_OUTPUT
   //    Q : Bool;
   // END_VAR
   // VAR
   //    Stat_Bit : Bool;
   // END_VAR
BEGIN
END_DATA_BLOCK

DATA_BLOCK "HourWork_DB_P1"   // DB5
AUTHOR : RTecmer
FAMILY : XMHour
VERSION : 0.1
// stored: AutoNumber true, DBAccessibleFromOPCUA true, InstanceOfName 09_W_Work counter, InstanceOfType FB
"09_W_Work counter"
BEGIN
END_DATA_BLOCK

DATA_BLOCK "HourWork_P4_DB"   // DB69
AUTHOR : RTecmer
FAMILY : XMHour
VERSION : 0.1
// stored: AutoNumber true, DBAccessibleFromOPCUA true, InstanceOfName 09_W_Work counter, InstanceOfType FB
"09_W_Work counter"
BEGIN
END_DATA_BLOCK

DATA_BLOCK "HourWork__P2_DB"   // DB14
AUTHOR : RTecmer
FAMILY : XMHour
VERSION : 0.1
// stored: AutoNumber true, DBAccessibleFromOPCUA true, InstanceOfName 09_W_Work counter, InstanceOfType FB
"09_W_Work counter"
BEGIN
END_DATA_BLOCK

DATA_BLOCK "HourWork__P3_DB"   // DB15
AUTHOR : RTecmer
FAMILY : XMHour
VERSION : 0.1
// stored: AutoNumber true, DBAccessibleFromOPCUA true, InstanceOfName 09_W_Work counter, InstanceOfType FB
"09_W_Work counter"
BEGIN
END_DATA_BLOCK

DATA_BLOCK "IEC_Counter_ControlAlarm_DB"   // DB73
{ S7_Optimized_Access := 'TRUE' }
// stored: AutoNumber false, DBAccessibleFromOPCUA true, InstanceOfName IEC_COUNTER, OfSystemLibElement IEC_COUNTER, OfSystemLibVersion 1.0
"IEC_COUNTER"
   // VAR RETAIN
   //    CU : Bool;
   //    CD : Bool;
   //    R : Bool;
   //    LD : Bool;
   //    QU : Bool;
   //    QD : Bool;
   //    PV : Int;
   //    CV : Int;
   // END_VAR
BEGIN
END_DATA_BLOCK

DATA_BLOCK "IEC_SetLimitFir1_0_DB"   // DB97
{ S7_Optimized_Access := 'TRUE' }
// stored: AutoNumber true, DBAccessibleFromOPCUA true, InstanceOfName IEC_TIMER, OfSystemLibElement IEC_TIMER, OfSystemLibVersion 1.0
"IEC_TIMER"
   // VAR
   //    PT : Time;
   //    ET { ExternalWritable := 'False'} : Time;
   //    IN : Bool;
   //    Q { ExternalWritable := 'False'} : Bool;
   // END_VAR
BEGIN
END_DATA_BLOCK

DATA_BLOCK "IEC_Timer1_Generator1Hz_DB"   // DB16
{ S7_Optimized_Access := 'TRUE' }
// stored: AutoNumber true, DBAccessibleFromOPCUA true, InstanceOfName IEC_TIMER, OfSystemLibElement IEC_TIMER, OfSystemLibVersion 1.0
"IEC_TIMER"
   // VAR
   //    PT : Time;
   //    ET { ExternalWritable := 'False'} : Time;
   //    IN : Bool;
   //    Q { ExternalWritable := 'False'} : Bool;
   // END_VAR
BEGIN
END_DATA_BLOCK

DATA_BLOCK "IEC_Timer2_Generator1Hz_DB"   // DB17
{ S7_Optimized_Access := 'TRUE' }
// stored: AutoNumber true, DBAccessibleFromOPCUA true, InstanceOfName IEC_TIMER, OfSystemLibElement IEC_TIMER, OfSystemLibVersion 1.0
"IEC_TIMER"
   // VAR
   //    PT : Time;
   //    ET { ExternalWritable := 'False'} : Time;
   //    IN : Bool;
   //    Q { ExternalWritable := 'False'} : Bool;
   // END_VAR
BEGIN
END_DATA_BLOCK

DATA_BLOCK "IEC_Timer_50Hz_DB"   // DB13
{ S7_Optimized_Access := 'TRUE' }
// stored: AutoNumber true, DBAccessibleFromOPCUA true, InstanceOfName IEC_TIMER, OfSystemLibElement IEC_TIMER, OfSystemLibVersion 1.0
"IEC_TIMER"
   // VAR
   //    PT : Time;
   //    ET { ExternalWritable := 'False'} : Time;
   //    IN : Bool;
   //    Q { ExternalWritable := 'False'} : Bool;
   // END_VAR
BEGIN
END_DATA_BLOCK

DATA_BLOCK "IEC_Timer_AlarmMagistrala_Niskie_DB"   // DB132
{ S7_Optimized_Access := 'TRUE' }
// stored: AutoNumber true, DBAccessibleFromOPCUA true, InstanceOfName IEC_TIMER, OfSystemLibElement IEC_TIMER, OfSystemLibVersion 1.0
"IEC_TIMER"
   // VAR
   //    PT : Time;
   //    ET { ExternalWritable := 'False'} : Time;
   //    IN : Bool;
   //    Q { ExternalWritable := 'False'} : Bool;
   // END_VAR
BEGIN
END_DATA_BLOCK

DATA_BLOCK "IEC_Timer_Ampere_Max_reset_DB"   // DB65
{ S7_Optimized_Access := 'TRUE' }
// stored: AutoNumber true, DBAccessibleFromOPCUA true, InstanceOfName IEC_TIMER, OfSystemLibElement IEC_TIMER, OfSystemLibVersion 1.0
"IEC_TIMER"
   // VAR
   //    PT : Time;
   //    ET { ExternalWritable := 'False'} : Time;
   //    IN : Bool;
   //    Q { ExternalWritable := 'False'} : Bool;
   // END_VAR
BEGIN
END_DATA_BLOCK

DATA_BLOCK "IEC_Timer_B7max_bar_DB"   // DB117
{ S7_Optimized_Access := 'TRUE' }
// stored: AutoNumber true, DBAccessibleFromOPCUA true, InstanceOfName IEC_TIMER, OfSystemLibElement IEC_TIMER, OfSystemLibVersion 1.0
"IEC_TIMER"
   // VAR
   //    PT : Time;
   //    ET { ExternalWritable := 'False'} : Time;
   //    IN : Bool;
   //    Q { ExternalWritable := 'False'} : Bool;
   // END_VAR
BEGIN
END_DATA_BLOCK

DATA_BLOCK "IEC_Timer_B7max_off_alarm_DB"   // DB142
{ S7_Optimized_Access := 'TRUE' }
// stored: AutoNumber true, DBAccessibleFromOPCUA true, InstanceOfName IEC_TIMER, OfSystemLibElement IEC_TIMER, OfSystemLibVersion 1.0
"IEC_TIMER"
   // VAR
   //    PT : Time;
   //    ET { ExternalWritable := 'False'} : Time;
   //    IN : Bool;
   //    Q { ExternalWritable := 'False'} : Bool;
   // END_VAR
BEGIN
END_DATA_BLOCK

DATA_BLOCK "IEC_Timer_Hist_SetHWork_P1_DB"   // DB43
{ S7_Optimized_Access := 'TRUE' }
// stored: AutoNumber true, DBAccessibleFromOPCUA true, InstanceOfName IEC_TIMER, OfSystemLibElement IEC_TIMER, OfSystemLibVersion 1.0
"IEC_TIMER"
   // VAR
   //    PT : Time;
   //    ET { ExternalWritable := 'False'} : Time;
   //    IN : Bool;
   //    Q { ExternalWritable := 'False'} : Bool;
   // END_VAR
BEGIN
END_DATA_BLOCK

DATA_BLOCK "IEC_Timer_Hist_SetHWork_P2_DB"   // DB44
{ S7_Optimized_Access := 'TRUE' }
// stored: AutoNumber true, DBAccessibleFromOPCUA true, InstanceOfName IEC_TIMER, OfSystemLibElement IEC_TIMER, OfSystemLibVersion 1.0
"IEC_TIMER"
   // VAR
   //    PT : Time;
   //    ET { ExternalWritable := 'False'} : Time;
   //    IN : Bool;
   //    Q { ExternalWritable := 'False'} : Bool;
   // END_VAR
BEGIN
END_DATA_BLOCK

DATA_BLOCK "IEC_Timer_Hist_SetHWork_P3_DB"   // DB45
{ S7_Optimized_Access := 'TRUE' }
// stored: AutoNumber true, DBAccessibleFromOPCUA true, InstanceOfName IEC_TIMER, OfSystemLibElement IEC_TIMER, OfSystemLibVersion 1.0
"IEC_TIMER"
   // VAR
   //    PT : Time;
   //    ET { ExternalWritable := 'False'} : Time;
   //    IN : Bool;
   //    Q { ExternalWritable := 'False'} : Bool;
   // END_VAR
BEGIN
END_DATA_BLOCK

DATA_BLOCK "IEC_Timer_Hist_SetHWork_P4_DB"   // DB28
{ S7_Optimized_Access := 'TRUE' }
// stored: AutoNumber true, DBAccessibleFromOPCUA true, InstanceOfName IEC_TIMER, OfSystemLibElement IEC_TIMER, OfSystemLibVersion 1.0
"IEC_TIMER"
   // VAR
   //    PT : Time;
   //    ET { ExternalWritable := 'False'} : Time;
   //    IN : Bool;
   //    Q { ExternalWritable := 'False'} : Bool;
   // END_VAR
BEGIN
END_DATA_BLOCK

DATA_BLOCK "IEC_Timer_HisterRresetNetwork50hz_DB"   // DB94
{ S7_Optimized_Access := 'TRUE' }
// stored: AutoNumber true, DBAccessibleFromOPCUA true, InstanceOfName IEC_TIMER, OfSystemLibElement IEC_TIMER, OfSystemLibVersion 1.0
"IEC_TIMER"
   // VAR
   //    PT : Time;
   //    ET { ExternalWritable := 'False'} : Time;
   //    IN : Bool;
   //    Q { ExternalWritable := 'False'} : Bool;
   // END_VAR
BEGIN
END_DATA_BLOCK

DATA_BLOCK "IEC_Timer_InputWarningH_DB"   // DB96
{ S7_Optimized_Access := 'TRUE' }
// stored: AutoNumber true, DBAccessibleFromOPCUA true, InstanceOfName IEC_TIMER, OfSystemLibElement IEC_TIMER, OfSystemLibVersion 1.0
"IEC_TIMER"
   // VAR
   //    PT : Time;
   //    ET { ExternalWritable := 'False'} : Time;
   //    IN : Bool;
   //    Q { ExternalWritable := 'False'} : Bool;
   // END_VAR
BEGIN
END_DATA_BLOCK

DATA_BLOCK "IEC_Timer_K1OFF_DB"   // DB11
{ S7_Optimized_Access := 'TRUE' }
// stored: AutoNumber true, DBAccessibleFromOPCUA true, InstanceOfName IEC_TIMER, OfSystemLibElement IEC_TIMER, OfSystemLibVersion 1.0
"IEC_TIMER"
   // VAR
   //    PT : Time;
   //    ET { ExternalWritable := 'False'} : Time;
   //    IN : Bool;
   //    Q { ExternalWritable := 'False'} : Bool;
   // END_VAR
BEGIN
END_DATA_BLOCK

DATA_BLOCK "IEC_Timer_K1ON_DB"   // DB12
{ S7_Optimized_Access := 'TRUE' }
// stored: AutoNumber true, DBAccessibleFromOPCUA true, InstanceOfName IEC_TIMER, OfSystemLibElement IEC_TIMER, OfSystemLibVersion 1.0
"IEC_TIMER"
   // VAR
   //    PT : Time;
   //    ET { ExternalWritable := 'False'} : Time;
   //    IN : Bool;
   //    Q { ExternalWritable := 'False'} : Bool;
   // END_VAR
BEGIN
END_DATA_BLOCK

DATA_BLOCK "IEC_Timer_K2OFF_DB"   // DB8
{ S7_Optimized_Access := 'TRUE' }
// stored: AutoNumber true, DBAccessibleFromOPCUA true, InstanceOfName IEC_TIMER, OfSystemLibElement IEC_TIMER, OfSystemLibVersion 1.0
"IEC_TIMER"
   // VAR
   //    PT : Time;
   //    ET { ExternalWritable := 'False'} : Time;
   //    IN : Bool;
   //    Q { ExternalWritable := 'False'} : Bool;
   // END_VAR
BEGIN
END_DATA_BLOCK

DATA_BLOCK "IEC_Timer_K2ON_DB"   // DB9
{ S7_Optimized_Access := 'TRUE' }
// stored: AutoNumber true, DBAccessibleFromOPCUA true, InstanceOfName IEC_TIMER, OfSystemLibElement IEC_TIMER, OfSystemLibVersion 1.0
"IEC_TIMER"
   // VAR
   //    PT : Time;
   //    ET { ExternalWritable := 'False'} : Time;
   //    IN : Bool;
   //    Q { ExternalWritable := 'False'} : Bool;
   // END_VAR
BEGIN
END_DATA_BLOCK

DATA_BLOCK "IEC_Timer_K3OFF_DB"   // DB26
{ S7_Optimized_Access := 'TRUE' }
// stored: AutoNumber true, DBAccessibleFromOPCUA true, InstanceOfName IEC_TIMER, OfSystemLibElement IEC_TIMER, OfSystemLibVersion 1.0
"IEC_TIMER"
   // VAR
   //    PT : Time;
   //    ET { ExternalWritable := 'False'} : Time;
   //    IN : Bool;
   //    Q { ExternalWritable := 'False'} : Bool;
   // END_VAR
BEGIN
END_DATA_BLOCK

DATA_BLOCK "IEC_Timer_K3ON_DB"   // DB25
{ S7_Optimized_Access := 'TRUE' }
// stored: AutoNumber true, DBAccessibleFromOPCUA true, InstanceOfName IEC_TIMER, OfSystemLibElement IEC_TIMER, OfSystemLibVersion 1.0
"IEC_TIMER"
   // VAR
   //    PT : Time;
   //    ET { ExternalWritable := 'False'} : Time;
   //    IN : Bool;
   //    Q { ExternalWritable := 'False'} : Bool;
   // END_VAR
BEGIN
END_DATA_BLOCK

DATA_BLOCK "IEC_Timer_P1_ready_DB"   // DB133
{ S7_Optimized_Access := 'TRUE' }
// stored: AutoNumber true, DBAccessibleFromOPCUA true, InstanceOfName IEC_TIMER, OfSystemLibElement IEC_TIMER, OfSystemLibVersion 1.0
"IEC_TIMER"
   // VAR
   //    PT : Time;
   //    ET { ExternalWritable := 'False'} : Time;
   //    IN : Bool;
   //    Q { ExternalWritable := 'False'} : Bool;
   // END_VAR
BEGIN
END_DATA_BLOCK

DATA_BLOCK "IEC_Timer_P2_ready_DB"   // DB144
{ S7_Optimized_Access := 'TRUE' }
// stored: AutoNumber true, DBAccessibleFromOPCUA true, InstanceOfName IEC_TIMER, OfSystemLibElement IEC_TIMER, OfSystemLibVersion 1.0
"IEC_TIMER"
   // VAR
   //    PT : Time;
   //    ET { ExternalWritable := 'False'} : Time;
   //    IN : Bool;
   //    Q { ExternalWritable := 'False'} : Bool;
   // END_VAR
BEGIN
END_DATA_BLOCK

DATA_BLOCK "IEC_Timer_P3_ready_DB"   // DB145
{ S7_Optimized_Access := 'TRUE' }
// stored: AutoNumber true, DBAccessibleFromOPCUA true, InstanceOfName IEC_TIMER, OfSystemLibElement IEC_TIMER, OfSystemLibVersion 1.0
"IEC_TIMER"
   // VAR
   //    PT : Time;
   //    ET { ExternalWritable := 'False'} : Time;
   //    IN : Bool;
   //    Q { ExternalWritable := 'False'} : Bool;
   // END_VAR
BEGIN
END_DATA_BLOCK

DATA_BLOCK "IEC_Timer_PressO2_Max_DB"   // DB63
{ S7_Optimized_Access := 'TRUE' }
// stored: AutoNumber true, DBAccessibleFromOPCUA true, InstanceOfName IEC_TIMER, OfSystemLibElement IEC_TIMER, OfSystemLibVersion 1.0
"IEC_TIMER"
   // VAR
   //    PT : Time;
   //    ET { ExternalWritable := 'False'} : Time;
   //    IN : Bool;
   //    Q { ExternalWritable := 'False'} : Bool;
   // END_VAR
BEGIN
END_DATA_BLOCK

DATA_BLOCK "IEC_Timer_ResK1errorRun_DB"   // DB101
{ S7_Optimized_Access := 'TRUE' }
// stored: AutoNumber true, DBAccessibleFromOPCUA true, InstanceOfName IEC_TIMER, OfSystemLibElement IEC_TIMER, OfSystemLibVersion 1.0
"IEC_TIMER"
   // VAR
   //    PT : Time;
   //    ET { ExternalWritable := 'False'} : Time;
   //    IN : Bool;
   //    Q { ExternalWritable := 'False'} : Bool;
   // END_VAR
BEGIN
END_DATA_BLOCK

DATA_BLOCK "IEC_Timer_ResetPID_stst0_DB"   // DB20
{ S7_Optimized_Access := 'TRUE' }
// stored: AutoNumber true, DBAccessibleFromOPCUA true, InstanceOfName IEC_TIMER, OfSystemLibElement IEC_TIMER, OfSystemLibVersion 1.0
"IEC_TIMER"
   // VAR
   //    PT : Time;
   //    ET { ExternalWritable := 'False'} : Time;
   //    IN : Bool;
   //    Q { ExternalWritable := 'False'} : Bool;
   // END_VAR
BEGIN
END_DATA_BLOCK

DATA_BLOCK "IEC_Timer_Reset_Is_Up_Hz_DB"   // DB50
{ S7_Optimized_Access := 'TRUE' }
// stored: AutoNumber true, DBAccessibleFromOPCUA true, InstanceOfName IEC_TIMER, OfSystemLibElement IEC_TIMER, OfSystemLibVersion 1.0
"IEC_TIMER"
   // VAR
   //    PT : Time;
   //    ET { ExternalWritable := 'False'} : Time;
   //    IN : Bool;
   //    Q { ExternalWritable := 'False'} : Bool;
   // END_VAR
BEGIN
END_DATA_BLOCK

DATA_BLOCK "IEC_Timer_Reset_Set_Motor2_DB"   // DB75
{ S7_Optimized_Access := 'TRUE' }
// stored: AutoNumber true, DBAccessibleFromOPCUA true, InstanceOfName IEC_TIMER, OfSystemLibElement IEC_TIMER, OfSystemLibVersion 1.0
"IEC_TIMER"
   // VAR
   //    PT : Time;
   //    ET { ExternalWritable := 'False'} : Time;
   //    IN : Bool;
   //    Q { ExternalWritable := 'False'} : Bool;
   // END_VAR
BEGIN
END_DATA_BLOCK

DATA_BLOCK "IEC_Timer_Reset_Set_Motor3_DB"   // DB93
{ S7_Optimized_Access := 'TRUE' }
// stored: AutoNumber true, DBAccessibleFromOPCUA true, InstanceOfName IEC_TIMER, OfSystemLibElement IEC_TIMER, OfSystemLibVersion 1.0
"IEC_TIMER"
   // VAR
   //    PT : Time;
   //    ET { ExternalWritable := 'False'} : Time;
   //    IN : Bool;
   //    Q { ExternalWritable := 'False'} : Bool;
   // END_VAR
BEGIN
END_DATA_BLOCK

DATA_BLOCK "IEC_Timer_Reset_Set_Motor4_DB"   // DB84
{ S7_Optimized_Access := 'TRUE' }
// stored: AutoNumber true, DBAccessibleFromOPCUA true, InstanceOfName IEC_TIMER, OfSystemLibElement IEC_TIMER, OfSystemLibVersion 1.0
"IEC_TIMER"
   // VAR
   //    PT : Time;
   //    ET { ExternalWritable := 'False'} : Time;
   //    IN : Bool;
   //    Q { ExternalWritable := 'False'} : Bool;
   // END_VAR
BEGIN
END_DATA_BLOCK

DATA_BLOCK "IEC_Timer_Reset_delay_DB"   // DB67
{ S7_Optimized_Access := 'TRUE' }
// stored: AutoNumber true, DBAccessibleFromOPCUA true, InstanceOfName IEC_TIMER, OfSystemLibElement IEC_TIMER, OfSystemLibVersion 1.0
"IEC_TIMER"
   // VAR
   //    PT : Time;
   //    ET { ExternalWritable := 'False'} : Time;
   //    IN : Bool;
   //    Q { ExternalWritable := 'False'} : Bool;
   // END_VAR
BEGIN
END_DATA_BLOCK

DATA_BLOCK "IEC_Timer_SUPV_SM_DB"   // DB95
{ S7_Optimized_Access := 'TRUE' }
// stored: AutoNumber true, DBAccessibleFromOPCUA true, InstanceOfName IEC_TIMER, OfSystemLibElement IEC_TIMER, OfSystemLibVersion 1.0
"IEC_TIMER"
   // VAR
   //    PT : Time;
   //    ET { ExternalWritable := 'False'} : Time;
   //    IN : Bool;
   //    Q { ExternalWritable := 'False'} : Bool;
   // END_VAR
BEGIN
END_DATA_BLOCK

DATA_BLOCK "IEC_Timer_Set_50Hz_DB"   // DB66
{ S7_Optimized_Access := 'TRUE' }
// stored: AutoNumber true, DBAccessibleFromOPCUA true, InstanceOfName IEC_TIMER, OfSystemLibElement IEC_TIMER, OfSystemLibVersion 1.0
"IEC_TIMER"
   // VAR
   //    PT : Time;
   //    ET { ExternalWritable := 'False'} : Time;
   //    IN : Bool;
   //    Q { ExternalWritable := 'False'} : Bool;
   // END_VAR
BEGIN
END_DATA_BLOCK

DATA_BLOCK "IEC_Timer_Set_Current_Overload_InverterKDN_DB"   // DB68
{ S7_Optimized_Access := 'TRUE' }
// stored: AutoNumber true, DBAccessibleFromOPCUA true, InstanceOfName IEC_TIMER, OfSystemLibElement IEC_TIMER, OfSystemLibVersion 1.0
"IEC_TIMER"
   // VAR
   //    PT : Time;
   //    ET { ExternalWritable := 'False'} : Time;
   //    IN : Bool;
   //    Q { ExternalWritable := 'False'} : Bool;
   // END_VAR
BEGIN
END_DATA_BLOCK

DATA_BLOCK "IEC_Timer_Start-InverterP2_DB"   // DB40
{ S7_Optimized_Access := 'TRUE' }
// stored: AutoNumber true, DBAccessibleFromOPCUA true, InstanceOfName IEC_TIMER, OfSystemLibElement IEC_TIMER, OfSystemLibVersion 1.0
"IEC_TIMER"
   // VAR
   //    PT : Time;
   //    ET { ExternalWritable := 'False'} : Time;
   //    IN : Bool;
   //    Q { ExternalWritable := 'False'} : Bool;
   // END_VAR
BEGIN
END_DATA_BLOCK

DATA_BLOCK "IEC_Timer_Start-InverterP3_DB"   // DB41
{ S7_Optimized_Access := 'TRUE' }
// stored: AutoNumber true, DBAccessibleFromOPCUA true, InstanceOfName IEC_TIMER, OfSystemLibElement IEC_TIMER, OfSystemLibVersion 1.0
"IEC_TIMER"
   // VAR
   //    PT : Time;
   //    ET { ExternalWritable := 'False'} : Time;
   //    IN : Bool;
   //    Q { ExternalWritable := 'False'} : Bool;
   // END_VAR
BEGIN
END_DATA_BLOCK

DATA_BLOCK "IEC_Timer_Start-InverterP4_DB"   // DB27
{ S7_Optimized_Access := 'TRUE' }
// stored: AutoNumber true, DBAccessibleFromOPCUA true, InstanceOfName IEC_TIMER, OfSystemLibElement IEC_TIMER, OfSystemLibVersion 1.0
"IEC_TIMER"
   // VAR
   //    PT : Time;
   //    ET { ExternalWritable := 'False'} : Time;
   //    IN : Bool;
   //    Q { ExternalWritable := 'False'} : Bool;
   // END_VAR
BEGIN
END_DATA_BLOCK

DATA_BLOCK "IEC_Timer_Start_InverterP1_DB"   // DB39
{ S7_Optimized_Access := 'TRUE' }
// stored: AutoNumber true, DBAccessibleFromOPCUA true, InstanceOfName IEC_TIMER, OfSystemLibElement IEC_TIMER, OfSystemLibVersion 1.0
"IEC_TIMER"
   // VAR
   //    PT : Time;
   //    ET { ExternalWritable := 'False'} : Time;
   //    IN : Bool;
   //    Q { ExternalWritable := 'False'} : Bool;
   // END_VAR
BEGIN
END_DATA_BLOCK

DATA_BLOCK "IEC_Timer_WatchDogWicc-PLC_DB"   // DB22
{ S7_Optimized_Access := 'TRUE' }
// stored: AutoNumber true, DBAccessibleFromOPCUA true, InstanceOfName IEC_TIMER, OfSystemLibElement IEC_TIMER, OfSystemLibVersion 1.0
"IEC_TIMER"
   // VAR
   //    PT : Time;
   //    ET { ExternalWritable := 'False'} : Time;
   //    IN : Bool;
   //    Q { ExternalWritable := 'False'} : Bool;
   // END_VAR
BEGIN
END_DATA_BLOCK

DATA_BLOCK "IEC_Timer_WatchDogWinCC_cd_DB"   // DB23
{ S7_Optimized_Access := 'TRUE' }
// stored: AutoNumber true, DBAccessibleFromOPCUA true, InstanceOfName IEC_TIMER, OfSystemLibElement IEC_TIMER, OfSystemLibVersion 1.0
"IEC_TIMER"
   // VAR
   //    PT : Time;
   //    ET { ExternalWritable := 'False'} : Time;
   //    IN : Bool;
   //    Q { ExternalWritable := 'False'} : Bool;
   // END_VAR
BEGIN
END_DATA_BLOCK

DATA_BLOCK "IEC_Timer_Z11_open_DB"   // DB89
{ S7_Optimized_Access := 'TRUE' }
// stored: AutoNumber true, DBAccessibleFromOPCUA true, InstanceOfName IEC_TIMER, OfSystemLibElement IEC_TIMER, OfSystemLibVersion 1.0
"IEC_TIMER"
   // VAR
   //    PT : Time;
   //    ET { ExternalWritable := 'False'} : Time;
   //    IN : Bool;
   //    Q { ExternalWritable := 'False'} : Bool;
   // END_VAR
BEGIN
END_DATA_BLOCK

DATA_BLOCK "IEC_Timer_Z11close_DB"   // DB131
{ S7_Optimized_Access := 'TRUE' }
// stored: AutoNumber true, DBAccessibleFromOPCUA true, InstanceOfName IEC_TIMER, OfSystemLibElement IEC_TIMER, OfSystemLibVersion 1.0
"IEC_TIMER"
   // VAR
   //    PT : Time;
   //    ET { ExternalWritable := 'False'} : Time;
   //    IN : Bool;
   //    Q { ExternalWritable := 'False'} : Bool;
   // END_VAR
BEGIN
END_DATA_BLOCK

DATA_BLOCK "IEC_Timer_alarm_reset_DB"   // DB98
{ S7_Optimized_Access := 'TRUE' }
// stored: AutoNumber true, DBAccessibleFromOPCUA true, InstanceOfName IEC_TIMER, OfSystemLibElement IEC_TIMER, OfSystemLibVersion 1.0
"IEC_TIMER"
   // VAR
   //    PT : Time;
   //    ET { ExternalWritable := 'False'} : Time;
   //    IN : Bool;
   //    Q { ExternalWritable := 'False'} : Bool;
   // END_VAR
BEGIN
END_DATA_BLOCK

DATA_BLOCK "IEC_Timer_errorRTU_histereza_DB"   // DB129
{ S7_Optimized_Access := 'TRUE' }
// stored: AutoNumber true, DBAccessibleFromOPCUA true, InstanceOfName IEC_TIMER, OfSystemLibElement IEC_TIMER, OfSystemLibVersion 1.0
"IEC_TIMER"
   // VAR
   //    PT : Time;
   //    ET { ExternalWritable := 'False'} : Time;
   //    IN : Bool;
   //    Q { ExternalWritable := 'False'} : Bool;
   // END_VAR
BEGIN
END_DATA_BLOCK

DATA_BLOCK "IEC_Timer_resDodtkowa_DB"   // DB111
{ S7_Optimized_Access := 'TRUE' }
// stored: AutoNumber true, DBAccessibleFromOPCUA true, InstanceOfName IEC_TIMER, OfSystemLibElement IEC_TIMER, OfSystemLibVersion 1.0
"IEC_TIMER"
   // VAR
   //    PT : Time;
   //    ET { ExternalWritable := 'False'} : Time;
   //    IN : Bool;
   //    Q { ExternalWritable := 'False'} : Bool;
   // END_VAR
BEGIN
END_DATA_BLOCK

DATA_BLOCK "IEC_Timer_resetAlarmMagistrala_Niskie_DB"   // DB137
{ S7_Optimized_Access := 'TRUE' }
// stored: AutoNumber true, DBAccessibleFromOPCUA true, InstanceOfName IEC_TIMER, OfSystemLibElement IEC_TIMER, OfSystemLibVersion 1.0
"IEC_TIMER"
   // VAR
   //    PT : Time;
   //    ET { ExternalWritable := 'False'} : Time;
   //    IN : Bool;
   //    Q { ExternalWritable := 'False'} : Bool;
   // END_VAR
BEGIN
END_DATA_BLOCK

DATA_BLOCK "IEC_Timer_tmp_up_reset_DB"   // DB140
{ S7_Optimized_Access := 'TRUE' }
// stored: AutoNumber true, DBAccessibleFromOPCUA true, InstanceOfName IEC_TIMER, OfSystemLibElement IEC_TIMER, OfSystemLibVersion 1.0
"IEC_TIMER"
   // VAR
   //    PT : Time;
   //    ET { ExternalWritable := 'False'} : Time;
   //    IN : Bool;
   //    Q { ExternalWritable := 'False'} : Bool;
   // END_VAR
BEGIN
END_DATA_BLOCK

DATA_BLOCK "MB_COMM_LOAD_DB"   // DB34
// stored: AutoNumber true, DBAccessibleFromOPCUA true, InstanceOfName MB_COMM_LOAD, OfSystemLibElement MB_COMM_LOAD, OfSystemLibVersion 2.1
"MB_COMM_LOAD"
   // VAR_INPUT
   //    REQ : Bool;
   //    PORT : PORT;
   //    BAUD : UDInt;
   //    PARITY : UInt;
   //    FLOW_CTRL : UInt;
   //    RTS_ON_DLY : UInt;
   //    RTS_OFF_DLY : UInt;
   //    RESP_TO : UInt;
   // END_VAR
   // VAR_OUTPUT
   //    DONE : Bool;
   //    ERROR : Bool;
   //    STATUS : Word;
   // END_VAR
   // VAR_IN_OUT
   //    MB_DB : MB_BASE;
   // END_VAR
   // VAR
   //    ICHAR_GAP : UInt;
   //    RETRIES : UInt;
   //    WRREC_STATUS : Word;
   //    RDREC_STATUS : Word;
   //    SFC_STATUS : Word;
   //    Port_CFG_SFB : Array[0..25] of Byte;
   //    Send_CFG_SFB : Array[0..16] of Byte;
   //    Rcv_CFG_SFB : Array[0..60] of Byte;
   //    STOP_BITS : USInt := 1;
   // END_VAR
BEGIN
END_DATA_BLOCK

DATA_BLOCK "MB_COMM_LOAD_DB_Slave1"   // DB127
// stored: AutoNumber true, DBAccessibleFromOPCUA true, InstanceOfName MB_COMM_LOAD, OfSystemLibElement MB_COMM_LOAD, OfSystemLibVersion 2.1
"MB_COMM_LOAD"
   // VAR_INPUT
   //    REQ : Bool;
   //    PORT : PORT;
   //    BAUD : UDInt;
   //    PARITY : UInt;
   //    FLOW_CTRL : UInt;
   //    RTS_ON_DLY : UInt;
   //    RTS_OFF_DLY : UInt;
   //    RESP_TO : UInt;
   // END_VAR
   // VAR_OUTPUT
   //    DONE : Bool;
   //    ERROR : Bool;
   //    STATUS : Word;
   // END_VAR
   // VAR_IN_OUT
   //    MB_DB : MB_BASE;
   // END_VAR
   // VAR
   //    ICHAR_GAP : UInt;
   //    RETRIES : UInt;
   //    WRREC_STATUS : Word;
   //    RDREC_STATUS : Word;
   //    SFC_STATUS : Word;
   //    Port_CFG_SFB : Array[0..25] of Byte;
   //    Send_CFG_SFB : Array[0..16] of Byte;
   //    Rcv_CFG_SFB : Array[0..60] of Byte;
   //    STOP_BITS : USInt;
   // END_VAR
BEGIN
END_DATA_BLOCK

DATA_BLOCK "MB_MASTER_DB"   // DB36
// stored: AutoNumber true, DBAccessibleFromOPCUA true, InstanceOfName MB_MASTER, OfSystemLibElement MB_MASTER, OfSystemLibVersion 2.2
"MB_MASTER"
   // // inherited from MB_BASE
   // VAR
   //    S_PORT : UInt;
   //    S_RESP_TO : UInt;
   //    S_ICHAR_GAP : UInt;
   //    S_RETRIES : UInt;
   // END_VAR
   // VAR_INPUT
   //    REQ : Bool;
   //    MB_ADDR : UInt;
   //    MODE : USInt;
   //    DATA_ADDR : UDInt;
   //    DATA_LEN : UInt;
   // END_VAR
   // VAR_OUTPUT
   //    DONE : Bool;
   //    BUSY : Bool;
   //    ERROR : Bool;
   //    STATUS : Word;
   // END_VAR
   // VAR_IN_OUT
   //    DATA_PTR : Variant;
   // END_VAR
   // VAR
   //    SEND_PTP_SFB : Array[0..11] of Byte;
   //    RCV_PTP_SFB : Array[0..11] of Byte;
   //    RCV_RST_SFB : Array[0..9] of Byte;
   //    PF_FREQUENCY : Real;
   //    BLOCKED_PROC_TIMEOUT : Real;
   //    CURRENT_TIME_VALUE : UDInt;
   //    SAVED_TIME_VALUE : UDInt;
   //    SAVED_SLAVE_ADDR : Word;
   //    SAVED_MODE : Word;
   //    SAVED_DATA_ADDR : DWord;
   //    SAVED_DATA_LEN : UInt;
   //    MB_STATE : UInt;
   //    COMM_SENT_COUNT : UInt;
   //    BYTE_COUNT : USInt;
   //    INIT_OK : Bool;
   //    ACTIVE : Bool;
   //    BROADCAST_FLAG : Bool;
   //    EXTENDED_ADDRESSING : Bool;
   //    SAVED_START_ADDR : UInt;
   //    TXBuf_Function_Offset : UDInt;
   //    TXBuf_Address_Offset : UDInt;
   //    TXBuf_Quantity_Offset : UDInt;
   // END_VAR
BEGIN
END_DATA_BLOCK

DATA_BLOCK "MB_SLAVE_RTU_DB"   // DB58
// stored: AutoNumber true, DBAccessibleFromOPCUA true, InstanceOfName MB_SLAVE, OfSystemLibElement MB_SLAVE, OfSystemLibVersion 2.1
"MB_SLAVE"
   // // inherited from MB_BASE
   // VAR
   //    S_PORT : UInt;
   //    S_RESP_TO : UInt;
   //    S_ICHAR_GAP : UInt;
   //    S_RETRIES : UInt;
   // END_VAR
   // VAR_INPUT
   //    MB_ADDR : UInt;
   // END_VAR
   // VAR_OUTPUT
   //    NDR : Bool;
   //    DR : Bool;
   //    ERROR : Bool;
   //    STATUS : Word;
   // END_VAR
   // VAR_IN_OUT
   //    MB_HOLD_REG : Variant;
   // END_VAR
   // VAR
   //    SEND_PTP_SFB : Array[0..11] of Byte;
   //    RCV_PTP_SFB : Array[0..11] of Byte;
   //    MB_State : Word;
   //    Request_Count : Word;
   //    Slave_Message_Count : Word;
   //    Bad_CRC_Count : Word;
   //    Broadcast_Count : Word;
   //    Exception_Count : Word;
   //    Success_Count : Word;
   //    SL_Status_Hold : Word;
   //    HR_Start_Offset : Word;
   //    Init_OK : Bool;
   //    Broadcast_Flag : Bool;
   //    SL_Error_State : Bool;
   //    Extended_Addressing : Bool;
   //    XMT_Set_NDR : Bool;
   //    XMT_Set_DR : Bool;
   // END_VAR
BEGIN
END_DATA_BLOCK

DATA_BLOCK "R_TRIG_DB_AUT_M1"   // DB118
// stored: AutoNumber true, DBAccessibleFromOPCUA true, InstanceOfName R_TRIG, OfSystemLibElement R_TRIG, OfSystemLibVersion 1.0
"R_TRIG"
   // VAR_INPUT
   //    CLK : Bool;
   // END_VAR
   // VAR_OUTPUT
   //    Q : Bool;
   // END_VAR
   // VAR
   //    Stat_Bit : Bool;
   // END_VAR
BEGIN
END_DATA_BLOCK

DATA_BLOCK "R_TRIG_DB_AUT_M2"   // DB120
// stored: AutoNumber true, DBAccessibleFromOPCUA true, InstanceOfName R_TRIG, OfSystemLibElement R_TRIG, OfSystemLibVersion 1.0
"R_TRIG"
   // VAR_INPUT
   //    CLK : Bool;
   // END_VAR
   // VAR_OUTPUT
   //    Q : Bool;
   // END_VAR
   // VAR
   //    Stat_Bit : Bool;
   // END_VAR
BEGIN
END_DATA_BLOCK

DATA_BLOCK "R_TRIG_DB_AUT_M3"   // DB121
// stored: AutoNumber true, DBAccessibleFromOPCUA true, InstanceOfName R_TRIG, OfSystemLibElement R_TRIG, OfSystemLibVersion 1.0
"R_TRIG"
   // VAR_INPUT
   //    CLK : Bool;
   // END_VAR
   // VAR_OUTPUT
   //    Q : Bool;
   // END_VAR
   // VAR
   //    Stat_Bit : Bool;
   // END_VAR
BEGIN
END_DATA_BLOCK

DATA_BLOCK "R_TRIG_DB_AUT_M4"   // DB122
// stored: AutoNumber true, DBAccessibleFromOPCUA true, InstanceOfName R_TRIG, OfSystemLibElement R_TRIG, OfSystemLibVersion 1.0
"R_TRIG"
   // VAR_INPUT
   //    CLK : Bool;
   // END_VAR
   // VAR_OUTPUT
   //    Q : Bool;
   // END_VAR
   // VAR
   //    Stat_Bit : Bool;
   // END_VAR
BEGIN
END_DATA_BLOCK

DATA_BLOCK "R_TRIG_DB_AUT_Z11"   // DB123
// stored: AutoNumber true, DBAccessibleFromOPCUA true, InstanceOfName R_TRIG, OfSystemLibElement R_TRIG, OfSystemLibVersion 1.0
"R_TRIG"
   // VAR_INPUT
   //    CLK : Bool;
   // END_VAR
   // VAR_OUTPUT
   //    Q : Bool;
   // END_VAR
   // VAR
   //    Stat_Bit : Bool;
   // END_VAR
BEGIN
END_DATA_BLOCK

DATA_BLOCK "R_TRIG_DB_CLK"   // DB126
// stored: AutoNumber true, DBAccessibleFromOPCUA true, InstanceOfName R_TRIG, OfSystemLibElement R_TRIG, OfSystemLibVersion 1.0
"R_TRIG"
   // VAR_INPUT
   //    CLK : Bool;
   // END_VAR
   // VAR_OUTPUT
   //    Q : Bool;
   // END_VAR
   // VAR
   //    Stat_Bit : Bool;
   // END_VAR
BEGIN
END_DATA_BLOCK

DATA_BLOCK "R_TRIG_DB_przechwycenie_strategii"   // DB138
// stored: AutoNumber true, DBAccessibleFromOPCUA true, InstanceOfName R_TRIG, OfSystemLibElement R_TRIG, OfSystemLibVersion 1.0
"R_TRIG"
   // VAR_INPUT
   //    CLK : Bool;
   // END_VAR
   // VAR_OUTPUT
   //    Q : Bool;
   // END_VAR
   // VAR
   //    Stat_Bit : Bool;
   // END_VAR
BEGIN
END_DATA_BLOCK

DATA_BLOCK "Strategia sterowania POMPOWNIA_DB"   // DB139
AUTHOR : rtecmer
VERSION : 0.1
// stored: AutoNumber true, DBAccessibleFromOPCUA true, InstanceOfName 06_M_Control strategy Pumping station, InstanceOfType FB
"06_M_Control strategy Pumping station"
BEGIN
END_DATA_BLOCK

DATA_BLOCK "ValueHz_in_Alarm_CurrentOver_DB"   // DB71
AUTHOR : rtecmer
VERSION : 0.1
// stored: AutoNumber true, DBAccessibleFromOPCUA true, InstanceOfName 06_M_Control Hz safe mode from bar Max, InstanceOfType FB
"06_M_Control Hz safe mode from bar Max"
BEGIN
END_DATA_BLOCK

DATA_BLOCK "dbByte Status P1P2P3P4_DB"   // DB77
AUTHOR : rtecmer
VERSION : 0.1
// stored: AutoNumber true, DBAccessibleFromOPCUA true, InstanceOfName 06_M_Byte status pomp, InstanceOfType FB
"06_M_Byte status pomp"
BEGIN
END_DATA_BLOCK

DATA_BLOCK "dbControl of   Inverters_DB"   // DB49
AUTHOR : rtecmer
VERSION : 0.1
// stored: AutoNumber true, DBAccessibleFromOPCUA true, InstanceOfName 06_M_Inverte control, InstanceOfType FB
"06_M_Inverte control"
BEGIN
END_DATA_BLOCK

DATA_BLOCK "dbControl of  connection Inverters_P2"   // DB51
AUTHOR : rtecmer
VERSION : 0.1
// stored: AutoNumber true, DBAccessibleFromOPCUA true, InstanceOfName 06_M_Inverter connection control, InstanceOfType FB
"06_M_Inverter connection control"
BEGIN
END_DATA_BLOCK

DATA_BLOCK "dbControl of  connection Inverters_P3"   // DB52
AUTHOR : rtecmer
VERSION : 0.1
// stored: AutoNumber true, DBAccessibleFromOPCUA true, InstanceOfName 06_M_Inverter connection control, InstanceOfType FB
"06_M_Inverter connection control"
BEGIN
END_DATA_BLOCK

DATA_BLOCK "dbControl of compressor conection network P2"   // DB53
AUTHOR : rtecmer
VERSION : 0.1
// stored: AutoNumber true, DBAccessibleFromOPCUA true, InstanceOfName 06_M_Network connection control, InstanceOfType FB
"06_M_Network connection control"
BEGIN
END_DATA_BLOCK

DATA_BLOCK "dbControl of compressor conection network"   // DB47
AUTHOR : rtecmer
VERSION : 0.1
// stored: AutoNumber true, DBAccessibleFromOPCUA true, InstanceOfName 06_M_Network connection control, InstanceOfType FB
"06_M_Network connection control"
BEGIN
END_DATA_BLOCK

DATA_BLOCK "dbControl of conection network_P1"   // DB54
AUTHOR : rtecmer
VERSION : 0.1
// stored: AutoNumber true, DBAccessibleFromOPCUA true, InstanceOfName 06_M_Network connection control, InstanceOfType FB
"06_M_Network connection control"
BEGIN
END_DATA_BLOCK

DATA_BLOCK "dbControl of conection network_P3"   // DB55
AUTHOR : rtecmer
VERSION : 0.1
// stored: AutoNumber true, DBAccessibleFromOPCUA true, InstanceOfName 06_M_Network connection control, InstanceOfType FB
"06_M_Network connection control"
BEGIN
END_DATA_BLOCK

DATA_BLOCK "dbControl of connection Inverters P1"   // DB42
AUTHOR : rtecmer
VERSION : 0.1
// stored: AutoNumber true, DBAccessibleFromOPCUA true, InstanceOfName 06_M_Inverter connection control, InstanceOfType FB
"06_M_Inverter connection control"
BEGIN
END_DATA_BLOCK

DATA_BLOCK "dbControl of connection Inverters P1_1"   // DB92
AUTHOR : rtecmer
VERSION : 0.1
// stored: AutoNumber true, DBAccessibleFromOPCUA true, InstanceOfName 06_M_Inverter connection control, InstanceOfType FB
"06_M_Inverter connection control"
BEGIN
END_DATA_BLOCK

DATA_BLOCK "dbControl press oxygen"   // DB64
AUTHOR : rtecmer
VERSION : 0.1
// stored: AutoNumber true, DBAccessibleFromOPCUA true, InstanceOfName 01_E_bar max, InstanceOfType FB
"01_E_bar max"
BEGIN
END_DATA_BLOCK

DATA_BLOCK "dbControl without inverter"   // DB76
AUTHOR : rtecmer
VERSION : 0.1
// stored: AutoNumber true, DBAccessibleFromOPCUA true, InstanceOfName 06_M_control without inverter, InstanceOfType FB
"06_M_control without inverter"
BEGIN
END_DATA_BLOCK

DATA_BLOCK "dbControll modors leading and extras"   // DB46
AUTHOR : rtecmer
VERSION : 0.1
// stored: AutoNumber true, DBAccessibleFromOPCUA true, InstanceOfName 06_M_Main and auxiliary pump, InstanceOfType FB
"06_M_Main and auxiliary pump"
BEGIN
END_DATA_BLOCK

DATA_BLOCK "dbSetup Write Parameters_KDN"   // DB62
AUTHOR : rtecmer
VERSION : 0.1
// stored: AutoNumber true, DBAccessibleFromOPCUA true, InstanceOfName 06_M_Initialization of start values, InstanceOfType FB
"06_M_Initialization of start values"
BEGIN
END_DATA_BLOCK

DATA_BLOCK "dbSterowanie dołaczaniem dodatkocych_FB1"   // DB3
AUTHOR : RTecmer
FAMILY : Ster
VERSION : 0.1
// stored: AutoNumber true, DBAccessibleFromOPCUA true, InstanceOfName 06_M_Control of switching on an additional pump, InstanceOfType FB
"06_M_Control of switching on an additional pump"
BEGIN
END_DATA_BLOCK

DATA_BLOCK "dbSterowanie dołączeniem falownika_P4"   // DB33
AUTHOR : rtecmer
VERSION : 0.1
// stored: AutoNumber true, DBAccessibleFromOPCUA true, InstanceOfName 06_M_Inverter connection control, InstanceOfType FB
"06_M_Inverter connection control"
BEGIN
END_DATA_BLOCK

DATA_BLOCK "dbSterowanie dołączeniem na sieć_P4"   // DB56
AUTHOR : rtecmer
VERSION : 0.1
// stored: AutoNumber true, DBAccessibleFromOPCUA true, InstanceOfName 06_M_Network connection control, InstanceOfType FB
"06_M_Network connection control"
BEGIN
END_DATA_BLOCK

DATA_BLOCK "dbValueHz_in_Alarm_Pressure_DB"   // DB70
AUTHOR : rtecmer
VERSION : 0.1
// stored: AutoNumber true, DBAccessibleFromOPCUA true, InstanceOfName 06_M_Control Hz safe mode from bar Max, InstanceOfType FB
"06_M_Control Hz safe mode from bar Max"
BEGIN
END_DATA_BLOCK

DATA_BLOCK "dbWatchDog HMI"   // DB60
AUTHOR : rtecmer
VERSION : 0.1
// stored: AutoNumber true, DBAccessibleFromOPCUA true, InstanceOfName 00_S_WatchDog HMI, InstanceOfType FB
"00_S_WatchDog HMI"
BEGIN
END_DATA_BLOCK

DATA_BLOCK "dbWatchDog PLC - WinCC"   // DB61
AUTHOR : rtecmer
VERSION : 0.1
// stored: AutoNumber true, DBAccessibleFromOPCUA true, InstanceOfName 00_S_WatchDog PLC - WinCC, InstanceOfType FB
"00_S_WatchDog PLC - WinCC"
BEGIN
END_DATA_BLOCK

DATA_BLOCK "dbcalculation_of_the_increment"   // DB18
AUTHOR : RTecmer
FAMILY : PID
VERSION : 0.1
// stored: AutoNumber true, DBAccessibleFromOPCUA true, InstanceOfName 07_E_Pressure build-up control, InstanceOfType FB
"07_E_Pressure build-up control"
BEGIN
END_DATA_BLOCK

DATA_BLOCK "filtr _kalmana_2_DB_1"   // DB128
VERSION : 0.1
// stored: AutoNumber true, DBAccessibleFromOPCUA true, InstanceOfName filtr _kalmana_2, InstanceOfType FB
"filtr _kalmana_2"
BEGIN
END_DATA_BLOCK

DATA_BLOCK "operating_mode_select_aut-man_DB"   // DB119
AUTHOR : rtecmer
VERSION : 0.1
// stored: AutoNumber true, DBAccessibleFromOPCUA true, InstanceOfName 08_C_operating_mode_select_aut-man, InstanceOfType FB
"08_C_operating_mode_select_aut-man"
BEGIN
END_DATA_BLOCK
